(* CoDeSys 2.3 library: Util_plc.lib *)

(* Global variable list: Globale_Variablen *)
(*
 PLC1131-Library with various Utility-Functions:
 1. Bit_xx:		BOOL-Array-Pack, -Split and -Scan
 2. Hwio_xx:	DWORD/DINT-Array-Pack and -Split
 3. Tcs_xx:	Interface to System-Time/Timer and Run-Time-System-Specials
 4. Util_xx:		String/Character-Handling
 5. Mem_xx:	Marker/Memory-Area-Handling
 6. MSys_xx:	Interface to Settings and Information from MCore/MSys
 Copyright: G.Bachmann GmbH, 1996-1997, Feldkirch - Austria
*)
VAR_GLOBAL CONSTANT
	UTIL_PLC_LIBVER			  :	STRING(16) 	:=	'V1.40 Release';	(* Version String *)
	UTIL_PLC_MMPREADY         : BOOL        :=  TRUE;               (* MMP Ready *)

    (* Error-Return-Codes *)
    Tcs_ERC_ParmInvalid:		DINT := -2;			(* Parameters are invalid *)
    Tcs_ERC_NoSelf:				DINT := -8;			(* Caller is no PLC *)
    Tcs_ERC_Internal:           DINT := -11;		(* external function not supported *)

    (* constants for 'AreaCode' of Mem_GetSize and Mem_Clear *)
    Tcs_MX_Code:				DINT := 1;
    Tcs_MB_Code:				DINT := 2;
    Tcs_MD_Code:				DINT := 3;
    Tcs_MR_Code:				DINT := 4;
    Tcs_MW_Code:				DINT := 5;
    Tcs_RD_Code:				DINT := 19;
    Tcs_GD_Code:				DINT := 35;

    (* these constants occur in 'ConfState' of TCS_ARGINFO *)
    Tcs_CONF_PassString:		DINT := 16#40;		(* ArgumentStr="..." *)
    Tcs_CONF_PassNumber:		DINT := 16#80;		(* ArgumentNum=... *)
    Tcs_CONF_ReinitRetain:		DINT := 16#400;
    Tcs_CONF_MarkerBattPool:	DINT := 16#800;
    Tcs_CONF_OverTime:			DINT := 16#1000;	(* RunTime > IntervalTime *)
    Tcs_CONF_SevereOverTime:	DINT := 16#2000;	(* RunTime >> IntervalTime *)

    (* constants for 'VersType' in Tcs_ARG_GetConfig' *)
	Tcs_VER_Alpha:                DINT := 1;          (* Alpha-Version *)
	Tcs_VER_Beta:                 DINT := 2;          (* Beta-Version *)
	Tcs_VER_Release:              DINT := 3;          (* Release-Version *)

    (* constants for 'DirCode' of MSys_GetDirName *)
    MSys_DIR_System:			DINT := 1;
    MSys_DIR_Driver:			DINT := 2;
    MSys_DIR_Application:		DINT := 3;
    MSys_DIR_Temporary:			DINT := 4;
    MSys_DIR_NonVolatile:		DINT := 5;

   (* constants for 'ProcType' of MSys_GetCpuInfo *)
    MSys_CPU_80386:				DINT := 0;			(* ME203/CS200/ES200 .. *)
    MSys_CPU_80486:				DINT := 1;
    MSys_CPU_Pentium:			DINT := 2;			(* MP2xx .. *)
	MSys_CPU_Geode: 			DINT := 3; 			(* AMD Geode *)
	MSys_CPU_Pentium3:			DINT := 4;			(* MPC2xx *)
	MSys_CPU_Pentium4: 			DINT := 5;
	MSys_CPU_Atom: 				DINT := 7;

	(* constants for 'RebootReason' of MSys_GetCpuInfo *)
	WDOG_REB_UNKNOWN: 			DINT := 0;			(* unknown reboot *)
	WDOG_REB_POWERFAIL: 		DINT := 1;			(* Powerfail caused reboot *)
	WDOG_REB_PANIC:				DINT := 2;			(* Panic caused reboot *)
	WDOG_REB_WDOGKNOWN:			DINT := 3;			(* Watchdog caused known reboot *)
	WDOG_REB_WDOGUNKNOWN:		DINT := 4;			(* unknown Watchdog reboot *)

	(* Return values of profile functions *)
	PF_E_PARM		: DINT := 16#800A_0110; (* invalid parameter *)
	PF_E_NOFILE		: DINT := 16#800A_0111; (* file not found *)
	PF_E_FILEBIG	: DINT := 16#800A_0112; (* file too big *)
	PF_E_FILEEMPTY	: DINT := 16#800A_0113; (* file is empty *)
	PF_E_NOSEC		: DINT := 16#800A_0114; (* section not found *)
	PF_E_NOGRP		: DINT := 16#800A_0115; (* group not found *)
	PF_E_NOKEY		: DINT := 16#800A_0116; (* keyword not found *)
	PF_E_ENDFILE	: DINT := 16#800A_0117; (* end of file reached *)
	PF_E_NOSET		: DINT := 16#800A_0119; (* set not found *)
	PF_E_NOUNIT		: DINT := 16#800A_0120; (* uint not found *)

	PF_MODE_RELOAD_FILE : DINT := 1; (* Reload configuration file on next read/write *)
	PF_MODE_USE_FILE : DINT := 2; (* Use configuration file (reset of PF_MODE_USE_DEFAULTS) *)
	PF_MODE_USE_DEFAULTS : DINT := 3; (* Use default values ignore configuration file *)
	PF_MODE_FILE_LOADED : DINT := 4; (* Use values from cache, do not load configuration file *)

	(* Commands of Util_CallCFcn *)
	Util_CMD_GetFcnHandle:			DWORD := 0;  (* get function handle *)
	Util_CMD_CallCFcn:				DWORD := 1;  (* call C-function *)

	(* State of Util_CallCFcn *)
	Util_ERR_CallC_HandleInit:			DINT := 1;  (* FB is not initialized *)
	Util_ERR_CallC_HandleOk:			DINT := 0;  (* able to call funcition handle *)
	Util_ERR_CallC_FcnNotFound:			DINT := -1;  (* function not found *)
	Util_ERR_CallC_NoHandle:			DINT := -2;  (* no function handle *)
	Util_ERR_CallC_InvalidCmd:			DINT := -3;  (* invalid command *)
	Util_ERR_CallC_NoSelf:				DINT := -8;	 (* caller is no PLC *)
    Util_ERR_CallC_Internal:            DINT := -11; (* internal error *)

	Util_CallC_Mode_C:					DINT := 0;	 (* native C function *)
	Util_CallC_Mode_PLC:				DINT := 1;	 (* PLC C function from external library *)

	(* possible states of Util_GetSymValByName and Util_SetSymValByName *)
	Util_ERR_SymVal_Ok:					DINT := 0;  (* success/no error *)
	Util_ERR_SymVal_InvalidName: 		DINT := -1; (* invalid/to long symbol-name *)
	Util_ERR_SymVal_NoHandle: 			DINT := -2; (* symbol not found in symbol-table *)
	Util_ERR_SymVal_InvalidLength: 		DINT := -3; (* an invalid symbol-values length *)

	(* possible errors of MSys_WdogSet *)
	Util_ERR_WDogSet_Ok: 				DINT := 0;	(* watchdog successfully reconfigured *)
	Util_ERR_WDogSet_WDNotActive:		DINT := -1;	(* watchdog has not been activated *)
	Util_ERR_WDogSet_LowWTime:			DINT := -2;	(* specified watch-time is too low *)
	Util_ERR_WDogSet_HighWTime:			DINT := -3; (* specified watch-time is too high *)
	Util_ERR_WDogSet_ConfigErr:			DINT := -4;	(* error configureing watch-dog *)

	(* Modes of Util_LIST_Get *)
	Util_LIST_GetHead:					DINT := 1; (* get head of list *)
	Util_LIST_GetTail:					DINT := 2; (* get tail of list *)
	Util_LIST_GetById:					DINT := 3; (* get a element by ID *)

	(* Modes of Util_LIST_Insert *)
	Util_LIST_InsertHead:				DINT := 1; (* insert a element at head *)
	Util_LIST_InsertTail:				DINT := 2; (* insert a element at tail *)

	(* Modes of Util_LIST_Remove *)
	Util_LIST_RemoveAll:				DINT := 0; (* remove all list elements *)
	Util_LIST_RemoveHead:				DINT := 1; (* remove head element *)
	Util_LIST_RemoveTail:				DINT := 2; (* remove tail element *)

	(* Error Codes of List FBs *)
	Util_ERR_LstOk:					DINT := 0;	(* Call was OK *)
	Util_ERR_LstNoMem:				DINT := -1; (* unable to alloc needed memory *)
	Util_ERR_LstInvHandle:			DINT := -2; (* invalid list handle *)
	Util_ERR_LstListEmpty:			DINT := -3; (* list is empty *)
	Util_ERR_LstListFull:			DINT := -4; (* list is full *)
	Util_ERR_LstInvCmd:				DINT := -5; (* invalid command *)
	Util_ERR_LstNotFound:			DINT := -6; (* list element was not found *)

	(* Modes of Util date and time functions *)
	Util_DT_Mode_UTC:			    DINT := 0; (* UTC time *)
	Util_DT_Mode_Local:			    DINT := 1; (* Local time *)

	(* Sources of Util_GetClock *)
	Util_CLOCK_RealTime: 			DINT := 0; (* system wide realtime clock *)
	Util_CLOCK_Monotonic: 			DINT := 16#1; (* Monotonic system-wide clock *)
	Util_CLOCK_Ptp: 				DINT := 16#10; (* PTP timer *)
	Util_CLOCK_RtcNano:				DINT := 16#20; (* RTC sec. + nanosec. based on CpuClocks,
													  since 3.95 same as CLOCK_REALTIME *)

	(* Results of Util64 timestamp functions *)
	Util64_TIMESTAMP_Result_OK:				DINT := 0; (* UTC time *)
	Util64_TIMESTAMP_Result_Error:			DINT := -1; (* Error, usually a struct pointer is NULL *)
	Util64_TIMESTAMP_Result_Overflow:		DINT := -2; (* overflow of 64bit value *)
	Util64_TIMESTAMP_Result_Underflow:		DINT := -3; (* underflow of 64bit value *)
	Util64_TIMESTAMP_Result_Negative:		DINT := -4; (* negative value *)
	Util64_TIMESTAMP_Result_Invalid_Range:	DINT := -5; (* range of parameter is invalid *)
	Util64_TIMESTAMP_Result_Zero:			DINT := -6; (* resulting value is 0 *)

END_VAR

(* Data type *)
(* return-structure of MSys_GetCpuInfo *)
TYPE MSYS_CPUINFO
STRUCT
	RetCode			: DINT;							(*  Success (0) - or Error-Code (<0) *)
	CpuSwitch		: DWORD;						(* Position/Code of Cpu-Switches *)
	ProcNum			: UDINT;						(* Processor-Number *)
	CpuClock		: UDINT;						(* Rate of Cpu-Clock in MHz *)
	TickRate		: UDINT;						(* Tick-Rate (Ticks per Second) for Scheduling *)
	TimeSlice		: UDINT;						(* Time-Slice in Ticks for Scheduling *)
	TotalTicks		: UDINT;						(* Number of Ticks since Power-Up *)
	AuxClkRate		: UDINT;						(* Rate of auxiliary Clock *)
	RestartCount	: UDINT;						(* Number of Restarts since last Reset of NV-Ram *)
	DebugMode		: DWORD;						(* DebugMode from MCONFIG.INI *)
	SizeDRam		: UDINT;						(* Size of 'Main'-Memory *)
	SizeNVRam		: UDINT;						(* Size of Non-Volatile-Ram *)
	ProcType		: UDINT;						(* Processor Type 0=80386, 2=Pentium *)
	pExtCpuInfo		: POINTER TO MSYS_EXTCPUINFO; 	(* Pointer to extended CPU info *)
	pEthStatist		: POINTER TO MSYS_ETHSTAT; 		(* Pointer to Ethernet statistik *)
	EnableMMP       : BOOL;                         (* M1 Multi Processing (SMP) enabled *)
    HyperThreading  : BOOL;                         (* Hyper threading active *)
    NbOfCores       : BYTE;                         (* Number OF logical cores available FOR SMP *)
    ReservedCores   : BYTE;                         (* Number OF reserved cores *)
END_STRUCT
END_TYPE

(* Data type *)
TYPE MSYS_ETHSTAT :
STRUCT
	InOverloadCount		: UDINT;					(* Counter input data overloads *)
	OutOverloadCount	: UDINT;					(* Counter output data overloads *)
	BcOverloadCount		: UDINT;					(* Counter broadcast overloads *)
	InBytes100msPeak	: UDINT;					(* In bytes peak load in 100 ms *)
	BcBytes100msPeak	: UDINT;					(* Broadcast peak load in 100 ms *)
	OutBytes100msPeak	: UDINT;					(* Out bytes peak load in 100 ms *)
	StartTicks10ms		: ARRAY[1..10] OF UDINT;	(* Ticks at start counting *)
	InBytes10ms			: ARRAY[1..10] OF UDINT;	(* In bytes last 10 millisec *)
	BcBytes10ms			: ARRAY[1..10] OF UDINT;	(* Broadcast bytes last 10 ms *)
	OutBytes10ms		: ARRAY[1..10] OF UDINT;	(* Out bytes last 10 millisec *)
	CurrIndex100s		: UDINT;					(* Index to xx100s[] 0 .. 9 *)
	InPacks100s			: ARRAY[1..10] OF UDINT;	(* In packets last 100 seconds *)
	InBytes100s			: ARRAY[1..10] OF UDINT;	(* In bytes last 100 seconds *)
	BcPacks100s			: ARRAY[1..10] OF UDINT;	(* Broadcast packets last 100 s *)
	BcBytes100s			: ARRAY[1..10] OF UDINT;	(* Broadcast bytes last 100 s *)
	OutPacks100s		: ARRAY[1..10] OF UDINT;	(* Out packets last 100 seconds *)
	OutBytes100s		: ARRAY[1..10] OF UDINT;	(* Out bytes last 100 seconds *)
	InPacksTotal		: UDINT;					(* In packets since reboot *)
	InBytesTotalLow		: DWORD;					(* In bytes since reboot low DWORD *)
	InBytesTotalHigh	: DWORD;					(* In bytes since reboot high DWORD *)
	BcPacksTotal		: UDINT;					(* Broadcasts since reboot *)
	BcBytesTotalLow		: DWORD;					(* Broadcast bytes since reboot low DWORD *)
	BcBytesTotalHigh	: DWORD;					(* Broadcast bytes since reboot high DWORD *)
	OutPacksTotal		: UDINT;					(* Out packets since reboot *)
	OutBytesTotalLow	: DWORD;					(* Out bytes since reboot low DWORD *)
	OutBytesTotalHigh	: DWORD;					(* Out bytes since reboot high DWORD *)
END_STRUCT
END_TYPE

(* Data type *)
TYPE MSYS_EXTCPUINFO :
STRUCT
	CurrTemp: UDINT; (* Current CPU temperature in % *)
	MinTemp: UDINT; (* Minimum CPU temperature in % *)
	MaxTemp: UDINT; (* Maximum CPU temperature in % *)
	CpuUsage100Low: DWORD; (* Cpu Usage last 100 seconds low DWord *)
	CpuUsage100High: DWORD; (* Cpu Usage last 100 seconds high DWord *)
	CpuUsage1000Low: DWORD; (* Cpu Usage last 1000 seconds low DWord *)
	CpuUsage1000High: DWORD; (* Cpu Usage last 1000 seconds high DWord *)
	CpuUsageTotalLow: DWORD; (* Accumulated Cpu Time in Clocks low DWord *)
	CpuUsageTotalHigh: DWORD; (* Accumulated Cpu Time in Clocks high DWord *)
	TotalTimeLow: DWORD; (* Clocks since last reset (100%) low DWord *)
	TotalTimeHigh: DWORD; (* Clocks since last reset (100%) high DWord *)
	Spare: ARRAY [1..4] OF UDINT; (* NOT used, 0 FOR now *)
	UnitsTime: UDINT; (* Clocks per us (CPU MHz) *)
	LastIdleTime: UDINT; (* TIME in us Idle last ran *)
	MaxPccErases: UDINT; (* Maximum PC-Card erases *)
	MaxFlashErases: UDINT; (* Maximum Flash erases *)
	StrayInterrupts: UDINT; (* Number of stray interrupts *)
	SyncHigh: UDINT; (* Sync Rate fuer High in us *)
	SyncLow: UDINT; (* Sync Rate fuer Low in us *)
	pSyncCount: POINTER TO UDINT; (* Sync interrupts since boot *)
	pAuxClkCount: POINTER TO UDINT; (* Aux clocks since boot *)
	PccPresent: BYTE; (* PC-Card is present *)
	PccPluggedIn: BYTE; (* PC-Card is plugged in *)
	PccWritable: BYTE; (* No PC-Card write protection *)
	PccCheckError: BYTE; (* Error in boot check on PC-Card *)
	FlashPresent: BYTE; (* File Flash is present *)
	FlashWritable: BYTE; (* No Flash write protection *)
	FlashCheckError: BYTE; (* Error in boot check on Flash *)
	NVRamSupplError: BYTE; (* Error in NV-Ram supply *)
	NVRamCheckError: BYTE; (* Error in boot check on NV-Ram *)
	StackCheckError: BYTE; (* Stack overflow in one task *)
	DRamCheckError: BYTE; (* Checksum error in DRam *)
	RTCError: BYTE; (* Error in RTC value *)
    SoftBootError: BYTE; (* Soft boot error, M1 BY run *)
    HardBootError: BYTE; (* Hard boot error, booting aborted *)
    LongNameEnable: BYTE; (* Long filenames ON/OFF *)
    TickSource: BYTE; (* M_TICK_TIMER, M_TICK_RTC *)
    SntpTimestamp: DATE; (* SNTP TIME in sec. since 1970 *)
    (* Below here needs MSys 2.00 Release *)
	RebootReason: UDINT; (* reboot reason *)
	RebootInf: STRING(39); (* reboot info text *)
    (* Below here needs MSys 3.20 Release *)
    SntpTimeRecv: TIMESPEC; (* Last received SNTP TIME *)
    SntpTimeCorr: TIMESPEC; (* Last received SNTP TIME maybe
                               corrected by "SntpMaxCorrection"
                               and converted to local time. *)
    SntpMaxCorrection: DWORD; (* Maximum allowed change per
                                 SNTP update [sec]. *)
END_STRUCT
END_TYPE

(* Data type *)
(* return-structure of  Tcs_ARG_GetConfig *)
TYPE TCS_ARGINFO
STRUCT
    Verbose: DINT;                   (* Verbose/Debug-Level *)
    StopAfterStart: DINT;            (* indicates loading by gb-PLC/PS *)
    ConfState: DWORD;                (* (see 'Global Constants') *)
    TimeSlice: DINT;                 (* Interval-Time in 0.1 Milli-Seconds *)
    WithWatchdog: DINT;              (* 1 if Watchdog supervision, 0 otherwise *)
    WatchTime: DINT;                 (* Watchdog-Time *)
    MissingModules: DWORD;           (* BitMask of missing modules (first 31 only) *)
    ArgNumber: DINT;                 (* Number of setting 'ArgumentNum=' *)
    ArgStringLen: DINT;              (* Len of String of setting 'ArgumentStr=' *)
    Name: STRING(15);                (* Name of running Project / Module *)
    VersCode: ARRAY[1..3] OF UDINT;  (* version of current project/sw-module *)
	VersType: UDINT;                 (* version type (see 'global constants') *)
END_STRUCT
END_TYPE

(* Data type *)
(* return-structure of Tcs_RTC_LocalTime and Tcs_RTC_UTCTime *)
(* date+time in this format can be converted back to type DATE_AND_TIME
    by Tcs_RTC_BuildDT *)
TYPE TCS_CLOCK
STRUCT
    Second: DINT;		(* range 0 - 59 *)
    Minute: DINT;		(* range 0 - 59 *)
    Hour: DINT;			(* range 0 - 23 *)
    Day: DINT;			(* range 1 - 31 *)
    Month: DINT;		(* range 1 - 12 *)
    Year: DINT;			(* years since 1900 *)
    WeekDay: DINT;	    (* range 0 = Sunday ... 6 = Saturday *)
    YearDay: DINT;		(* range 0 - 365 *)
    DSTFlag: DINT;		(* DayLightSaving-Time Flag *)
END_STRUCT
END_TYPE

(* Data type *)
(* return-structure of Tcs_CYC_GetCycStat *)
TYPE TCS_CYCSTAT
STRUCT						(* all times in this structure are in ticks *)
    EntrySize: DINT;		(* size of this structure in bytes *)
    EntryType: DINT;		(* scaling of times to ticks (ticks per 0.1 Milli-Second) *)
    Running: DINT;			(* scaling of times to ticks (tick-duration in 0.1 Milli-Seconds *)
    Priority: DINT;			(* specified task priority *)
    CycTime: DWORD;			(* specified Interval-Time *)
    DiffTime: DWORD;		(* period between last two cycle-starts *)
    MinTime: DWORD;			(* min. DiffTime seen *)
    MaxTime: DWORD;			(* max. DiffTime seen *)
    AvgTime: DWORD;			(* average of DiffTime *)
    AvgParam: DWORD;		(* 32 *)
    CycCnt: DWORD;			(* counter of cycles *)
    Activity: DWORD;		(* reserved *)
    LastTime: DWORD;		(* time-stamp of last cycle *)
    MinRunTime: DWORD;		(* (only computed if CycTime > 0): min. of period of cycles *)
    MaxRunTime: DWORD;		(* (only computed if CycTime > 0): max. of period of cycles *)
    AvgRunTime: DWORD;		(* (only computed if CycTime > 0): avg. of period of cycles *)
	Running_us: DWORD;		(* tick-duration in micro-seconds, needs MSYS 2.02 or above *)
END_STRUCT
END_TYPE

(* Data type *)
TYPE TIMESPEC :
STRUCT
	DateAndTime: DT;
    NanoSeconds: UDINT;
END_STRUCT
END_TYPE

(* Data type *)
(* 64bit Timestamp split into DATE, TIME and NanoSeconds *)
TYPE UTIL64_DATETIME :
STRUCT
	DateValue  : DATE; (* DATE part of 64bit Timestamp *)
	TimeValue : TIME; (* TIME part of 64bit Timestamp *)
	NanoSeconds : UDINT; (* Nanosecons not contained in TimeValue *)
END_STRUCT
END_TYPE

(* Data type *)
(* 64bit Timestamp Value for time in nanoseconds *)
(* The value is unsigned *)
TYPE UTIL64_TIMESTAMP :
STRUCT
	TimestampNsLow  : DWORD; (* 4 byte little endian low part of 64bit *)
	TimestampNsHigh : DWORD; (* 4 byte little endian high part of 64bit *)
END_STRUCT
END_TYPE

(* Data type *)
(* return-structure of Util_GetCycStat *)
TYPE UTIL_CYCSTAT :
STRUCT
    Priority: DINT;			(* specified task priority [vxworks] *)
    CycTime: DWORD;			(* specified cycle-time [us] *)
	MainRatio: DWORD;		(* execution-rate of the task-POU *)
    CycCnt: DWORD;			(* counter of cycles *)
    RunTimeMin: DWORD;		(* Minimum Run Time in us *)
    RunTimeMax: DWORD;		(* Maximum Run Time in us *)
    RunTimeAvg: DWORD;		(* Average Run Time in us *)
	RunTimeTotal: DWORD;	(* Total run time in us *)
	CycleTimeMin: DWORD;    (* Minimum Cycle TIME in us *)
    CycleTimeMax: DWORD;    (* Maximum Cycle TIME in us *)
    CycleTimeAvg: DWORD;    (* Average Cycle TIME in us *)
	ErrorCode:  DINT;		(* OK/Done, Error-Code in case of error *)
END_STRUCT
END_TYPE

(* Data type *)
(* time structure TM *)
(* this time structure can be converted to DATE_AND_TIME (DT) *)
TYPE UTIL_TM
STRUCT
    Second: DINT;		(* range 0 - 59 *)
    Minute: DINT;		(* range 0 - 59 *)
    Hour: DINT;			(* range 0 - 23 *)
    Day: DINT;			(* range 1 - 31 *)
    Month: DINT;		(* range 1 - 12 *)
    Year: DINT;			(* years since 1900 *)
    WeekDay: DINT;	    (* range 0 = Sunday ... 6 = Saturday *)
    YearDay: DINT;		(* range 0 - 365 *)
    DSTFlag: DINT;		(* DayLightSaving-Time Flag *)
END_STRUCT
END_TYPE

(* POU BCD_TO_DINT, ST *)
(******************************************************************************
Description: Converts from BCD to Integer(32bit)
Input:
  - Num: BCD-value; Range 8 digits
Output:
    none
Return:
    Integer(32bit) value of BCD-value: Range 0 to 99999999
******************************************************************************)
FUNCTION BCD_TO_DINT : DINT
VAR_INPUT
	Num : DWORD;
END_VAR
;
END_FUNCTION

(* POU BCD_TO_INT, ST *)
(******************************************************************************
Description: Converts from BCD to Integer(16bit)
Input:
  - Num: BCD-value; Range 4 digits
Output:
    none
Return:
    Integer(16bit) value of BCD-value: Range 0 to 9999
******************************************************************************)
FUNCTION BCD_TO_INT : INT
VAR_INPUT
	Num : WORD;
END_VAR
;
END_FUNCTION

(* POU BCD_TO_SINT, ST *)
(******************************************************************************
Description: Converts from BCD to Integer(8bit)
Input:
  - Num: BCD-value; Range 2 digits
Output:
    none
Return:
    Integer(8bit) value of BCD-value: Range 0 to 99
******************************************************************************)
FUNCTION BCD_TO_SINT : SINT
VAR_INPUT
	Num : BYTE;
END_VAR
;
END_FUNCTION

(* POU Bit_FieldPack, IL *)
(******************************************************************************
Description: Packs Bits of the BOOL-Array to a DWORD-Array
Input:
  - StartAddrBits: Address of the BOOL array, use ADR() operator
  - StartIndx: Start index
  - EndIndx: End index
  - BitsTogether: Determines the number of Bits to pack together in a DWORD 
  - StartAddrPacked: Address of the DWORD-Array, use ADR() operator
Output:
  - StartAddrPacked: Moved bits from BOOL-Array
Return: Function checks if 'EndIndx'+1-'StartIndx' must is multiple 
    of 'BitsTogether'!
    - TRUE: Parameters are OK
    - FALSE: Wrong parameters
******************************************************************************)
FUNCTION Bit_FieldPack : BOOL
VAR_INPUT
	StartAddrBits: DWORD;
	StartIndx: DINT;
	EndIndx: DINT;
	BitsTogether: DINT;
	StartAddrPacked: DWORD;
END_VAR
	LD		0
END_FUNCTION

(* POU Bit_FieldScan, IL *)
(******************************************************************************
Description: Scans the BOOL-Array from StartIndx to EndIndx for the 
    first TRUE-Element
Input:
  - StartAddr: Address of BOOL array, use ADR() operator
  - StartIndx: Start index
  - EndIndx: End index
Output:
    none
Return: Index of the first TRUE element, or all zero
    - >= 0: Index of element
    - -1: no TRUE element is found
******************************************************************************)
FUNCTION Bit_FieldScan : DINT
VAR_INPUT
	StartAddr: DWORD;
	StartIndx: DINT;
	EndIndx: DINT;
END_VAR
LD 0
END_FUNCTION

(* POU Bit_FieldScanPack, IL *)
(******************************************************************************
Description: Packs Bits of the BOOL-Array to a DWORD-Array and scans for the
	last RUE element
Input:
  - StartAddrBits: Address of the BOOL array, use ADR() operator
  - StartIndx: Start index
  - EndIndx: End index
  - BitsTogether: Determines the number of Bits to pack together in a DWORD 
  - StartAddrPacked: Address of the DWORD-Array, use ADR() operator
Output:
  - StartAddrPacked: Moved bits from BOOL-Array
Return: Function checks if 'EndIndx'+1-'StartIndx' must is multiple 
    of 'BitsTogether'!
    - -2: Parameters are not OL
    - -1: No TRUE element is found
    - >= 0: Index of the last TRUE element
******************************************************************************)
FUNCTION Bit_FieldScanPack : DINT
VAR_INPUT
	StartAddrBits: DWORD;
	StartIndx: DINT;
	EndIndx: DINT;
	BitsTogether: DINT;
	StartAddrPacked: DWORD;
END_VAR
LD 0
END_FUNCTION

(* POU Bit_Pack, IL *)
(******************************************************************************
Description: Packs Bits of the BOOL-Array into a DWORD
Input:
  - StartAddr: Address of the BOOL array, use ADR() operator
  - NumberOf: Number of packing bits
Output:
    none
Return: Packed infomation of BOOL-array
*******************************************************************************)
FUNCTION Bit_Pack : DWORD
VAR_INPUT
	StartAddr: DWORD;
	NumberOf: DINT;
END_VAR
LD 0
END_FUNCTION

(* POU Bit_Split, IL *)
(******************************************************************************
Description: Unpacks Bits of a DWORD into a BOOL-Array
Input:
  - StartAddr: Address of the BOOL array, use ADR() operator
  - NumberOf: Number of depacking bits beginning at 0
  - Value: Packed Bits
Output:
  - StartAddr: This BOOL-array contains the unpacked bits of the DWORD
Return: Count equal to the set bits of the 'NumberOf'-Bits
*******************************************************************************)
FUNCTION Bit_Split : DINT
VAR_INPUT
	StartAddr: DWORD;
	NumberOf: DINT;
	Value: DWORD;
END_VAR
LD 0
END_FUNCTION

(* POU DINT_TO_BCD, ST *)
(******************************************************************************
Description: Converts from Integer(32bit) to BCD
Input:
  - Num: Integer(32bit) value; Range 0 to 99999999
Output:
    none
Return:
    BCD value; Range 8 digits
******************************************************************************)
FUNCTION DINT_TO_BCD : DWORD
VAR_INPUT
	Num : DINT;
END_VAR
;
END_FUNCTION

(* POU Hwio_Pack16, IL *)
(******************************************************************************
Description: Packs 16 values (type must be DWORD/DINT!) [set/clear] between 
    'StartAddr' and 'EndAddr' into a WORD (16bit)
Input:
  - StartAddr: Start address, use ADR() operator
  - EndAddr: End address, use ADR() operator
Output:
    none 
Return: WORD with packed bits
******************************************************************************)
FUNCTION Hwio_Pack16 : WORD
VAR_INPUT
    StartAddr: DWORD;
    EndAddr: DWORD; 
END_VAR
LD FALSE
END_FUNCTION

(* POU Hwio_Pack32, IL *)
(******************************************************************************
Description: Packs 32 values (type must be DWORD/DINT!) [set/clear] between 
    'StartAddr' and 'EndAddr' into a DWORD (32bit)
Input:
  - StartAddr: Start address, use ADR() operator
  - EndAddr: End address, use ADR() operator
Output:
    none 
Return: DWORD with packed bits
******************************************************************************)
FUNCTION Hwio_Pack32 : DWORD
VAR_INPUT
    StartAddr: DWORD;
    EndAddr: DWORD; 
END_VAR
LD FALSE
END_FUNCTION

(* POU Hwio_Pack8, IL *)
(******************************************************************************
Description: Packs 8 values (type must be DWORD/DINT!) [set/clear] between 
    'StartAddr' and 'EndAddr' into a DWORD (8bit)
Input:
  - StartAddr: Start address, use ADR() operator
  - EndAddr: End address, use ADR() operator
Output:
    none 
Return: BYTE with packed bits
******************************************************************************)
FUNCTION Hwio_Pack8 : BYTE
VAR_INPUT
    StartAddr: DWORD;
    EndAddr: DWORD; 
END_VAR
LD FALSE
END_FUNCTION

(* POU Hwio_Unpack, IL *)
(******************************************************************************
Description: Unpacking bits of a DWORD into a field of DWORDs [set/clear] 
Input:
  - StartAddr: Start address, use ADR() operator
  - EndAddr: End address, use ADR() operator
  - NumberOf: Number of unpacking bits
  - Packed: Value with packed bits
Output:
  - StartAddr to EndAddr: Unpacked bits
Return: If operation succeded
  - 0: Successful
  - Tcs_ERC_ParmInvalid: 'NumberOf' exceeds elements between 'Start'- 
    and 'EndAddr' 
******************************************************************************)
FUNCTION Hwio_Unpack : DINT
VAR_INPUT
    Packed: DWORD;  
    StartAddr: DWORD;
    EndAddr: DWORD; 
    NumberOf: DINT; 
END_VAR
LD FALSE
END_FUNCTION

(* POU INT_TO_BCD, ST *)
(******************************************************************************
Description: Converts from Integer(16bit) to BCD
Input:
  - Num: Integer(32bit) value; Range 0 to 9999
Output:
    none
Return:
    BCD value; Range 4 digits
******************************************************************************)
FUNCTION INT_TO_BCD : WORD
VAR_INPUT
	Num : INT;
END_VAR
;
END_FUNCTION

(* POU M100_PWMDutyCycleConv, ST *)
(******************************************************************************
Description: Converts a DutyCycle REAL to UINT.    
Input:
  - DutyCycle: with percent float value in range 0...100%
               Not fitting values will be limited to the valid range.
Output:
    none
Return:
	UINT converted DutyCycle. Value range. 0 .. 32768 (equals 100%)
******************************************************************************)
FUNCTION M100_PWMDutyCycleConv : WORD
VAR_INPUT
    DutyCycle : REAL;
END_VAR
;
END_FUNCTION

(* POU M100IO_GetCountedEvent, ST *)
(******************************************************************************
Description: splits a CountedEvent in its parts
Input:
  - Value: the current CountedEvent value to be split
Output:
  - State: state of the Event
  - Counter: how many times the event occured
  - NewEvent: true if the Counter changed since the last FB call
******************************************************************************)
FUNCTION_BLOCK M100IO_GetCountedEvent
VAR_INPUT
    Value : BYTE;
END_VAR
VAR_OUTPUT
	State : BOOL;
	Counter : WORD;
	NewEvent : BOOL;
END_VAR
VAR
	LastCounter : WORD;
END_VAR
;
END_FUNCTION_BLOCK

(* POU Mem_AtomicCopy, IL *)
(******************************************************************************
Description: Copy Memory-Area1 (Src) to Memory-Area2 (Dst) consistenly. All 
             reading and writing participants must use this function for a 
		     protection. 

Input:
  - Dst: Destination adress = Startadress of Memory-Area2
  - Src: Source adress = Start-adress of Memory-Area1 
  - Len: Length of the Memory-Area
Output:
    none 
Return: 
  - 0: Successful
  - Tcs_ERC_NoSelf: Caller is no PLC
  - Tcs_ERC_ParmInvalid: Parameters are invalid
******************************************************************************)
FUNCTION Mem_AtomicCopy : DINT
VAR_INPUT
	Dst: UDINT;
	Src: UDINT;
	Len: UDINT;
END_VAR
	LD		0
END_FUNCTION

(* POU Mem_Clear, IL *)
(******************************************************************************
Description: Clears the Memory/Marker-Area specified by 'AreaCode'
Input:
  - AreaCode: see CONSTANT variables Tcs_XX_Code, only this values are allowed
Output:
    none 
Return: Number of elements in the Area or error code
  - >= 0: Number of elements in the Area
  - -2: 'AreaCode' is invalid 
******************************************************************************)
FUNCTION Mem_Clear : DINT
VAR_INPUT
	AreaCode: DINT;
END_VAR
LD 0
END_FUNCTION

(* POU Mem_Copy, IL *)
(******************************************************************************
Description: Copy Memory-Area1 (Src) to Memory-Area2 (Dst)
Input:
  - Src: Source adress = Start-adress of Memory-Area1 
  - Dst: Destination adress = Startadress of Memory-Area2
  - Len: Length of the Memory-Area
Output:
    none 
Return: 
  -  0: Successful
  - -8: Caller is no PLC
******************************************************************************)
FUNCTION Mem_Copy : DINT
VAR_INPUT
	Dst: UDINT;
	Src: UDINT;
	Len: UDINT;
END_VAR
	LD		0
END_FUNCTION

(* POU Mem_GetSize, IL *)
(******************************************************************************
Description: Number of elements in the Memory/Marker-Area
Input:
  - AreaCode: see CONSTANT variables Tcs_xx_Code, only this values are allowed
Output:
    none 
Return: Number of elements in the Area or error code
  - >= 0: Number of elements in the Memory/Marker-Area
  - -2: 'AreaCode' is invalid 
******************************************************************************)
FUNCTION Mem_GetSize : DINT
VAR_INPUT
	AreaCode: DINT;
END_VAR
LD 0
END_FUNCTION

(* POU MSys_GetCpuInfo, IL *)
(******************************************************************************
Description: Fetching the system structure MSYS_CPUINFO
Input:
  - Dummy: meaningless
Output:
    none
Return:
    System structure MSYS_CPUINFO (see description in data types)
******************************************************************************)
FUNCTION MSys_GetCpuInfo : MSYS_CPUINFO
VAR_INPUT
	Dummy: DINT;
END_VAR
LD 0
END_FUNCTION

(* POU MSys_GetDirName, IL *)
(******************************************************************************
Description: Returns the path of the directory
Input:
  - DirCode: Code of directory
Output:
    none
Return:
    String of the system directory
******************************************************************************)
FUNCTION MSys_GetDirName : STRING(255)
VAR_INPUT
	DirCode: DINT;
END_VAR
LD 0
END_FUNCTION

(* POU MSys_GoPanic, ST *)
(******************************************************************************
Description: Initiate a System-Panic (SYS_APPPANIC)
Input:
  - Dummy: meaningless
Output:
    none
Return:
    meaningless
******************************************************************************)
FUNCTION MSys_GoPanic : DINT
VAR_INPUT
	Dummy: DINT;
END_VAR
;
END_FUNCTION

(* POU MSys_WdogSet, ST *)
(******************************************************************************
Description: reconfigures the watch-time of a projects software watch-dog,
             the watch-dog must have been activated

Note: be careful with applying a watch-time, 
	  the watch-time must have an adequate relation to the cycle-time and
      can cause reboots through the watch-dog if configured too low. 

Input:
  - WatchTime: watchdog-time, in milli- or micro-seconds
  - IsMicro: 0 - watch-time is in milli-seconds, 
             1 - watch-time is in micro-seconds
Return:
    zero on success or error-number otherwise
******************************************************************************)
FUNCTION MSys_WdogSet : DINT
VAR_INPUT
	WatchTime: UDINT;
	IsMicro: BOOL;
END_VAR
VAR
END_VAR
;
END_FUNCTION

(* POU MSys_WdogTrigger, ST *)
(******************************************************************************
Description: Trigger the software-watchdog of the PLC-project 
Input:
  - Dummy: meaningless
Output:
    none
Return:
    meaningless
******************************************************************************)
FUNCTION MSys_WdogTrigger : DINT
VAR_INPUT
	Dummy: DINT;
END_VAR
;
END_FUNCTION

(* POU Pf_Control, ST *)
(******************************************************************************
Description: Sets a specific mode of the Pf_Get and Pf_Set functions.    
Input:
  - Cmnd: mode to set (PF_MODE_XX)
Output:
    none
Return:
	>= 0 OK, line number (beginning at 0)
	< 0...error, see VAR_CONSTANT PF_E_XXX; convert this values with 
          DWORD_TO_DINT()
******************************************************************************)
FUNCTION Pf_Control : DINT
VAR_INPUT
	Cmnd	: DINT;
END_VAR
VAR
END_VAR
;
END_FUNCTION

(* POU pf_GetBool, ST *)
(******************************************************************************
Description: Reads a boolean value out of the specified file. Expression of 
    value in file has to be ON, OFF, YES, NO, TRUE, FALSE, 1 or 0. 
    Use this function in init section of PLC, it can take a little bit.    
Input:
  - Section: Name of section, 15 characters are significant, case sensitive. 
             If the string is empty it is used as a wildcard. 
  - Group: Name of group, 15 characters are significant, case sensitive. 
           If the string is empty it is used as a wildcard. 
  - Keyword: Name of keyword, 15 characters are significant, case sensitive
  - Default: Default Value, written to value when Keyword not found
  - Value: Returned value, use ADR() operator
  - StartLine: Start line of searching
  - FileName: file name, if an empty string is passed then in 'mconfig.ini' is searched
Output:
    none
Return:
	>= 0 OK, line number (beginning at 0)
	< 0...error, see VAR_CONSTANT PF_E_XXX; convert this values with 
          DWORD_TO_DINT()
******************************************************************************)
FUNCTION pf_GetBool : DINT
VAR_INPUT
	Section		: STRING;
	Group		: STRING;
	Keyword		: STRING;
	Default		: DINT;
	Value		: POINTER TO DINT;
	StartLine	: DINT;
	FileName	: STRING;
END_VAR
VAR
END_VAR
;
END_FUNCTION

(* POU pf_GetBoolExt, ST *)
(******************************************************************************
Description: Reads a boolean value out of the specified file. Expression of 
    value in file has to be ON, OFF, YES, NO, TRUE, FALSE, 1 or 0. 
    Use this function in init section of PLC, it can take a little bit.    
Input:
  - Section: 	Name of section, 15 characters are significant, case sensitive. 
             	If the string is empty it is used as a wildcard. 
  - Group: 		Name of group, 15 characters are significant, case sensitive. 
           	 	If the string is empty it is used as a wildcard. 
  - Set:     	Name of set, 15 characters are significant, case sensitive. 
             	If the string is empty it is used as a wildcard. 
  - Unit: 	 	Name of unit, 15 characters are significant, case sensitive. 
           	 	If the string is empty it is used as a wildcard. 
  - Keyword: 	Name of keyword, 15 characters are significant, case sensitive
  - Default: 	Default Value, written to value when Keyword not found
  - Value: 	 	Returned value, use ADR() operator
  - StartLine: 	Start line of searching
  - FileName: 	File name, if an empty string is passed then 'mconfig.ini' is used
Output:
    none
Return:
	>= 0 OK, line number (beginning at 0)
	< 0...error, see VAR_CONSTANT PF_E_XXX; convert this values with 
          DWORD_TO_DINT()
******************************************************************************)
FUNCTION pf_GetBoolExt : DINT
VAR_INPUT
	Section		: STRING;
	Group		: STRING;
	Set			: STRING;
	Unit		: STRING;
	Keyword		: STRING;
	Default		: DINT;
	Value		: POINTER TO DINT;
	StartLine	: DINT;
	FileName	: STRING;
END_VAR
VAR
END_VAR
;
END_FUNCTION

(* POU pf_GetInt, IL *)
(******************************************************************************
Description: Reads an integer value out of the specified file. 
    Use this function in init section of PLC, it can take a little bit.    
Input:
  - Section: Name of section, 15 characters are significant, case sensitive. 
             If the string is empty it is used as a wildcard. 
  - Group: Name of group, 15 characters are significant, case sensitive. 
           If the string is empty it is used as a wildcard. 
  - Keyword: Name of keyword, 15 characters are significant, case sensitive
  - Default: Default Value, written to value when Keyword not found
  - Value: Returned value, use ADR() operator
  - StartLine: Start line of searching
  - FileName: file name, if an empty string is passed then in 'mconfig.ini' is searched
Output:
    none
Return:
	>= 0 OK, line number (beginning at 0)
	< 0...error, see VAR_CONSTANT PF_E_XXX; convert this values with 
          DWORD_TO_DINT()
******************************************************************************)
FUNCTION pf_GetInt : DINT
VAR_INPUT
	Section		: STRING;
	Group		: STRING;
	Keyword		: STRING;
	Default		: DINT;
	Value		: POINTER TO DINT;
	StartLine	: DINT;
	FileName	: STRING;
END_VAR
VAR
END_VAR
	LD		0
END_FUNCTION

(* POU pf_GetIntExt, IL *)
(******************************************************************************
Description: Reads an integer value out of the specified file. 
    Use this function in init section of PLC, it can take a little bit.    
Input:
  - Section: 	Name of section, 15 characters are significant, case sensitive. 
             	If the string is empty it is used as a wildcard. 
  - Group: 		Name of group, 15 characters are significant, case sensitive. 
           	 	If the string is empty it is used as a wildcard. 
  - Set:     	Name of set, 15 characters are significant, case sensitive. 
             	If the string is empty it is used as a wildcard. 
  - Unit: 	 	Name of unit, 15 characters are significant, case sensitive. 
           	 	If the string is empty it is used as a wildcard. 
  - Keyword: 	Name of keyword, 15 characters are significant, case sensitive
  - Default: 	Default Value, written to value when Keyword not found
  - Value: 	 	Returned value, use ADR() operator
  - StartLine: 	Start line of searching
  - FileName: 	File name, if an empty string is passed then 'mconfig.ini' is used
Output:
    none
Return:
	>= 0 OK, line number (beginning at 0)
	< 0...error, see VAR_CONSTANT PF_E_XXX; convert this values with 
          DWORD_TO_DINT()
******************************************************************************)
FUNCTION pf_GetIntExt : DINT
VAR_INPUT
	Section		: STRING;
	Group		: STRING;
	Set			: STRING;
	Unit		: STRING;
	Keyword		: STRING;
	Default		: DINT;
	Value		: POINTER TO DINT;
	StartLine	: DINT;
	FileName	: STRING;
END_VAR
VAR
END_VAR
	LD		0
END_FUNCTION

(* POU pf_GetSecGrp, ST *)
(******************************************************************************
Description: returns the name of the preceding section and group of the passed-on
             line number. 

Input:
  - LastLine: the search starts from this line backwards. 
  - FileName: file name, if an empty string is passed then in 'mconfig.ini' is searched
Output:
  - Section: Name of section, 15 characters are significant, case sensitive
  - Group: Name of group, 15 characters are significant, case sensitive 
Return:
	>= 0 OK, line number (beginning at 0)
	< 0...error, see VAR_CONSTANT PF_E_XXX; convert this values with 
          DWORD_TO_DINT()
******************************************************************************)

FUNCTION pf_GetSecGrp : DINT
VAR_INPUT
	Section: STRING(15);
	Group: STRING(15);
	LastLine: DINT;
	FileName: STRING;
END_VAR
VAR
END_VAR
;
END_FUNCTION

(* POU Pf_GetStrg, ST *)
(******************************************************************************
Description: Reads a string value out of the specified file. 
    Use this function in init section of PLC, it can take a little bit.    
Input:
  - Section: Name of section, 15 characters are significant, case sensitive. 
             If the string is empty it is used as a wildcard. 
  - Group: Name of group, 15 characters are significant, case sensitive. 
           If the string is empty it is used as a wildcard. 
  - Keyword: Name of keyword, 15 characters are significant, case sensitive
  - Default: Default Value, written to value when Keyword not found  
  - Value: Returned value, max 80 characters
		   Important: String size has to be 80 chars !!
  - StartLine: Start line of searching
  - FileName: file name, if an empty string is passed then in 'mconfig.ini' is searched
Output:
    none
Return:
	>= 0 OK, line number (beginning at 0)
	< 0...error, see VAR_CONSTANT PF_E_XXX; convert this values with 
          DWORD_TO_DINT()
******************************************************************************)
FUNCTION Pf_GetStrg : DINT
VAR_INPUT
	Section		: STRING;
	Group		: STRING;
	Keyword		: STRING;
	Default		: STRING;
	Value		: STRING;
	StartLine	: DINT;
	FileName	: STRING;
END_VAR
VAR
END_VAR
;
END_FUNCTION

(* POU Pf_GetStrg2, ST *)
(******************************************************************************
Description: Reads a string value out of the specified file.
	This is the same function as Pf_GetStrg except for the max length of the 
    value sting.  
    Use this function in init section of PLC, it can take a little bit.    
Input:
  - Section: Name of section, 15 characters are significant, case sensitive. 
             If the string is empty it is used as a wildcard. 
  - Group: Name of group, 15 characters are significant, case sensitive. 
           If the string is empty it is used as a wildcard. 
  - Keyword: Name of keyword, 15 characters are significant, case sensitive
  - Default: Default Value, written to value when Keyword not found
  - Value: Returned value (not a default string)
		   Since M-Base 3.70 149 characters are supported. The maximum length of 
           Pf_GetStr2 is reduced by the length of the keyword and of the string " = ".
		   Important: String size has to be 255 chars !!
  - StartLine: Start line of searching
  - FileName: file name, if an empty string is passed then in 'mconfig.ini' is searched
Output:
    none
Return:
	>= 0 OK, line number (beginning at 0)
	< 0...error, see VAR_CONSTANT PF_E_XXX; convert this values with 
          DWORD_TO_DINT()
******************************************************************************)
FUNCTION Pf_GetStrg2 : DINT
VAR_INPUT
	Section		: STRING;
	Group		: STRING;
	Keyword		: STRING;
	Default		: STRING;
	Value		: STRING(255);
	StartLine	: DINT;
	FileName	: STRING;
END_VAR
VAR
END_VAR
;
END_FUNCTION

(* POU Pf_GetStrgExt, ST *)
(******************************************************************************
Description: Reads a string value out of the specified file. 
    Use this function in init section of PLC, it can take a little bit.    
Input:
  - Section: 	Name of section, 15 characters are significant, case sensitive. 
             	If the string is empty it is used as a wildcard. 
  - Group: 		Name of group, 15 characters are significant, case sensitive. 
           	 	If the string is empty it is used as a wildcard. 
  - Set:     	Name of set, 15 characters are significant, case sensitive. 
             	If the string is empty it is used as a wildcard. 
  - Unit: 	 	Name of unit, 15 characters are significant, case sensitive. 
           	 	If the string is empty it is used as a wildcard. 
  - Keyword: 	Name of keyword, 15 characters are significant, case sensitive
  - Default: 	Default Value, written to value when Keyword not found
  - Value: 	 	Returned value, use ADR() operator. 
                Important: String size has to be 255 chars !!
                Since M-Base 3.70 149 characters are supported. The maximum length of 
                Pf_GetStrgExt is reduced by the length of the keyword and of the string 
                " = ".
  - StartLine: 	Start line of searching
  - FileName: 	File name, if an empty string is passed then 'mconfig.ini' is used
Output:
    none
Return:
	>= 0 OK, line number (beginning at 0)
	< 0...error, see VAR_CONSTANT PF_E_XXX; convert this values with 
          DWORD_TO_DINT()
******************************************************************************)
FUNCTION Pf_GetStrgExt : DINT
VAR_INPUT
	Section		: STRING;
	Group		: STRING;
	Set			: STRING;
	Unit		: STRING;
	Keyword		: STRING;
	Default		: STRING;
	Value		: STRING(255);
	StartLine	: DINT;
	FileName	: STRING;
END_VAR
VAR
END_VAR
;
END_FUNCTION

(* POU Pf_SetStrg_NB, ST *)
(******************************************************************************
Description: Writes a string value in the specified file. The keywords value 
             can be edited only, it must exist already. This is a non-blocking 
             function. 
Input:
  - Req:  request-enable
  - Section: Name of section, 15 characters are significant, case sensitive. 
             If the string is empty it is used as a wildcard. 
  - Group: Name of group, 15 characters are significant, case sensitive. 
           If the string is empty it is used as a wildcard. 
  - Keyword: Name of keyword, 15 characters are significant, case sensitive
  - Value: value, max 255 characters (the Core components of MBASE 3.50 support 
           max. 80 characters for the whole line of the keyword entry).
		   Since M-Base 3.70 149 characters are supported. The maximum length of 
           Pf_SetStrg_NB is reduced by the length of the keyword and of the string " = ".
  - StartLine: Start line of searching
  - FileName: file name, if an empty string is passed then in 'mconfig.ini' is searched
Output:
  - Done:  TRUE => operation completed 
  - Error:  TRUE in case of error 
  - Status:  0: OK/Done, 1: BUSY, Error-Code in case of error 
    (see VAR_CONSTANT PF_E_XXX; convert this values with DWORD_TO_DINT())
  - WrittenLine: written line number (beginning at 0)

******************************************************************************)
FUNCTION_BLOCK Pf_SetStrg_NB
VAR_INPUT
	Req         : BOOL;
	Section     : STRING;
	Group       : STRING;
	Keyword		: STRING;
	Value       : STRING(255);
	StartLine   : DINT;
	FileName    : STRING;
END_VAR
VAR_OUTPUT
	Done        : BOOL;
	Error       : BOOL;
	Status      : DINT;
    WrittenLine : UDINT;
END_VAR
VAR
    Pltd        : DWORD;
END_VAR
;
END_FUNCTION_BLOCK

(* POU Pf_SetStrgExt_NB, ST *)
(******************************************************************************
Description: Writes a string value in the specified file. The keywords value 
             can be edited only, it must exist already. This is a non-blocking 
             function. 
Input:
  - Req:  		request-enable
  - Section: 	Name of section, 15 characters are significant, case sensitive. 
             	If the string is empty it is used as a wildcard. 
  - Group: 		Name of group, 15 characters are significant, case sensitive. 
           	 	If the string is empty it is used as a wildcard. 
  - Set:     	Name of set, 15 characters are significant, case sensitive. 
             	If the string is empty it is used as a wildcard. 
  - Unit: 	 	Name of unit, 15 characters are significant, case sensitive. 
           	 	If the string is empty it is used as a wildcard. 
  - Keyword: 	Name of keyword, 15 characters are significant, case sensitive
  - Value: 		value, max 255 characters (the Core components of MBASE 3.50 support 
           		max. 80 characters for the whole line of the keyword entry)
 		        Since M-Base 3.70 149 characters are supported. The maximum length of 
                Pf_SetStrgExt_NB is reduced by the length of the keyword and of the 
                string " = ".
  - StartLine: 	Start line of search
  - FileName: 	file name, if an empty string is passed then 'mconfig.ini' is used
Output:
  - Done:  		TRUE => operation completed 
  - Error:  	TRUE in case of error 
  - Status:  	0: OK/Done, 1: BUSY, Error-Code in case of error 
			    (see VAR_CONSTANT PF_E_XXX; convert this values with DWORD_TO_DINT())
  - WrittenLine: written line number (beginning at 0)

******************************************************************************)
FUNCTION_BLOCK Pf_SetStrgExt_NB
VAR_INPUT
	Req         : BOOL;
	Section     : STRING;
	Group       : STRING;
	Set			: STRING;
	Unit		: STRING;
	Keyword		: STRING;
	Value       : STRING(255);
	StartLine   : DINT;
	FileName    : STRING;
END_VAR
VAR_OUTPUT
	Done        : BOOL;
	Error       : BOOL;
	Status      : DINT;
    WrittenLine : UDINT;
END_VAR
VAR
    Pltd        : DWORD;
END_VAR
;
END_FUNCTION_BLOCK

(* POU RTC_GetClock, ST *)
(******************************************************************************
Description: Gets the current time value of the system clock.
             This routine returns the system clock in seconds since 1970-01-01.
             The returned value is either UTC or LOCAL time, depending on 
             configured system time base.

Input:
  - Dummy: meaningless
Output:
    none
Return:
  - TIMESPEC structure (seconds + nanosecond part)
******************************************************************************)

FUNCTION RTC_GetClock : TIMESPEC
VAR_INPUT
	dummy: BOOL;
END_VAR
VAR
END_VAR
;
END_FUNCTION

(* POU SINT_TO_BCD, ST *)
(******************************************************************************
Description: Converts from Integer(8bit) to BCD
Input:
  - Num: Integer(32bit) value; Range 0 to 99
Output:
    none
Return:
    BCD value; Range 2 digits
******************************************************************************)
FUNCTION SINT_TO_BCD : BYTE
VAR_INPUT
	Num : SINT;
END_VAR
;
END_FUNCTION

(* POU Tcs_ARG_GetArgString, IL *)
(******************************************************************************
Description: Returns the String set with 'ArgumentStr=' (see file MCONFIG.INI)
Input:
  - Dummy: meaningless
Output:
    none
Return:
    String of Parameter 'ArgumentStr=' in file MCONFIG.INI
******************************************************************************)
FUNCTION Tcs_ARG_GetArgString : STRING(255)
VAR_INPUT
    Dummy: DINT;
END_VAR
LD FALSE
END_FUNCTION

(* POU Tcs_ARG_GetConfig, IL *)
(******************************************************************************
Description: Returns the system structure TCS_ARGINFO 
Input:
  - Dummy: meaningless
Output:
    none
Return:
    System Structure TCS_ARGINFO of current CPU (not all fields meaningful)
*****************************************************************************)
FUNCTION Tcs_ARG_GetConfig : TCS_ARGINFO
VAR_INPUT
    Dummy: DINT;
END_VAR
LD FALSE
END_FUNCTION

(* POU Tcs_CYC_GetCycStat, IL *)
(******************************************************************************
Description: Gets a copy of CYCSTAT-data. Deprecated support for the 
             first-task only since multitasking-environment (MSYS 3.80 R). 
             Multitasking is supported by Util_GetCycStat(). 
Input:
  - Dummy: meaningless
Output:
    none
Return:
  - TCS_CYCSTAT structure
******************************************************************************)
FUNCTION Tcs_CYC_GetCycStat: TCS_CYCSTAT
VAR_INPUT
    Dummy: DINT;
END_VAR
	LD		FALSE
END_FUNCTION

(* POU Tcs_CYC_GetMainRatio, IL *)
(******************************************************************************
Description: Returns Ratio of Intervals of Cyclic-Task(PLC_TASK) and SPS-Cycle. 
             Deprecated support for the first-task only since multitasking- 
             environment (MSYS 3.80 R). Multitasking is supported by 
             Util_GetCycStat(). 
Input:
  - Dummy: meaningless
Output:
    none
Return:
  - Tcs_CYC_GetMainRatio structure
******************************************************************************)
FUNCTION Tcs_CYC_GetMainRatio: DINT
VAR_INPUT
    Dummy: DINT;
END_VAR
	LD		FALSE
END_FUNCTION

(* POU Tcs_CYC_ReinitCycStat, IL *)
(******************************************************************************
Description: Reinit CYCSTAT-data
Input:
  - Dummy: meaningless
Output:
    none
Return:
    meaningless
******************************************************************************)
FUNCTION Tcs_CYC_ReinitCycStat: DINT
VAR_INPUT
    Dummy: DINT;
END_VAR
	LD		FALSE
END_FUNCTION

(* POU Tcs_CYC_SetCycStat, IL *)
(******************************************************************************
Description: Sets CYCSTAT/INTERVAL-data. Deprecated support for the 
             first-task only since multitasking-environment (MSYS 3.80 R).
             Multitasking is supported by Util_SetCycStat(). 
Input:
  - CycTime: PLC Interval Time in Ticks 
  - MainRatio: Ratio of PLC Interval Time to Task Interval Time
  - Priority: VxWorks Priority between 16 and 255
Output:
    none
Return: 
    meaningless
******************************************************************************)
FUNCTION Tcs_CYC_SetCycStat: DINT
VAR_INPUT
    CycTime: DWORD;
    MainRatio: DINT;
    Priority: DINT;
END_VAR
	LD		FALSE
END_FUNCTION

(* POU Tcs_EXC_Check, IL *)
(******************************************************************************
Description: Test Exception-Restart
Input:
  - Dummy: meaningless
Output:
    none
Return: Result of Exception-Restart
  - 1: Exception-Restart has been performed
  - else: not performed
*****************************************************************************)
FUNCTION Tcs_EXC_Check: DINT
VAR_INPUT
    Dummy: DINT;
END_VAR
LD FALSE
END_FUNCTION

(* POU Tcs_OLC_Check, IL *)
(******************************************************************************
Description: Test if an online change has been performed
Input:
  - Dummy: meaningless
Output:
    none
Return: Result of testing online change
  - 1: Online change has been performed
  - else: not performed
*****************************************************************************)
FUNCTION Tcs_OLC_Check: DINT
VAR_INPUT
    Dummy: DINT;
END_VAR
LD FALSE
END_FUNCTION

(* POU Tcs_RTC_BuildDT, IL *)
(******************************************************************************
Description: Converts TCS_CLOCK to DT-value according to local time zone
Input:
  - Clock: Time in format of TCS_CLOCK
Output:
    none
Return: 
    Time of format DATE_AND_TIME 
******************************************************************************)
FUNCTION Tcs_RTC_BuildDT: DATE_AND_TIME
VAR_INPUT
    Clock: TCS_CLOCK;
END_VAR
LD FALSE
END_FUNCTION

(* POU Tcs_RTC_GetDateAndTime, IL *)
(******************************************************************************
Description: Gets the current system date & time.
             This routine returns the current system time in either UTC or 
             LOCAL time, depending on configured system time base.

             ATTENTION: This function is deprecated. Please use 
                        function Util_RTC_GetDateAndTime instead 
                        of this function.

Input:
  - Dummy: meaningless
Output:
    none
Return: 
    Current date and time in DATE_AND_TIME format
******************************************************************************)
FUNCTION Tcs_RTC_GetDateAndTime: DATE_AND_TIME
VAR_INPUT
    Dummy: DINT;
END_VAR
LD FALSE
END_FUNCTION

(* POU Tcs_RTC_GetTime, IL *)
(******************************************************************************
Description: Get a monotonous time in microsecond resolution.
             This routine returns 'm_GetProcTime()' internally.
Input:
  - Dummy: meaningless
Output:
    none
Return: 
    Monotonous time
******************************************************************************)
FUNCTION Tcs_RTC_GetTime : UDINT
VAR_INPUT
    Dummy: DINT;
END_VAR
LD FALSE
END_FUNCTION

(* POU Tcs_RTC_LocalTime, IL *)
(******************************************************************************
Description: Converts DT to TCS_CLOCK according to local time zone
             (the local time-zone is considered since MSYS 3.10 R and 
             a compatibility-mode of >= 3.10)

             ATTENTION: This function is deprecated. Please use 
                        function Util_RTC_GetDateAndTime instead 
                        of this function.

Input:
  - D: Time of format DATE_AND_TIME
Output:
    none
Return: 
    Structure TCS_CLOCK
******************************************************************************)
FUNCTION Tcs_RTC_LocalTime: TCS_CLOCK
VAR_INPUT
    D: DATE_AND_TIME;
END_VAR
	LD		FALSE
END_FUNCTION

(* POU Tcs_RTC_SetDateAndTime, IL *)
(******************************************************************************
Description: Sets the current system date & time.
             This routine sets the system time to the value specified. Given
             time represents UTC or LOCAL time, depending on configured system
             timebase.

             ATTENTION: This function is deprecated. Please use 
                        function Util_RTC_SetDateAndTime instead 
                        of this function.

Input:
  - D: Date and Time of format DATE_AND_TIME 
Output:
    none
Return: Info of the action
  - 0: OK
  - 1: BUSY
  - else: ErrorCode
******************************************************************************)
FUNCTION Tcs_RTC_SetDateAndTime: DINT
VAR_INPUT
    D: DATE_AND_TIME;
END_VAR
LD FALSE
END_FUNCTION

(* POU Tcs_RTC_UTCTime, IL *)
(******************************************************************************
Description: Converts DT to TCS_CLOCK according to universal time zone (UTC)

             ATTENTION: This function is deprecated. Please use 
                        function Util_RTC_GetDateAndTime instead 
                        of this function.

Input:
  - D: Date and Time of format DATE_AND_TIME 
Output:
    none
Return: 
    Date and Time of format TCS_CLOCK
******************************************************************************)
FUNCTION Tcs_RTC_UTCTime: TCS_CLOCK
VAR_INPUT
    D: DATE_AND_TIME; 
END_VAR
LD FALSE
END_FUNCTION

(* POU Util64_ARRAY_TO_TIMESTAMP, ST *)
(******************************************************************************
Description: Converts from BYTE ARRAY[1..8] to 64bit Timestamp.    
Input:
  - TimestampNs: 8 Byte Array with little endian Timestamp raw data
  - TimestampResult: pointer to UTIL64_TIMESTAMP structure to be filled with
                     the result
Output:
    none
Return: DINT
	 0: Success (Util64_TIMESTAMP_Result_OK)
	-1: Error (Util64_TIMESTAMP_Result_Error)
	-6: timestamp is 0 (Util64_TIMESTAMP_Result_Zero)
******************************************************************************)
FUNCTION Util64_ARRAY_TO_TIMESTAMP : DINT
VAR_INPUT
	TimestampNs : ARRAY[1..8] OF BYTE;
	TimestampResult : POINTER TO UTIL64_TIMESTAMP;
END_VAR
;
END_FUNCTION

(* POU Util64_DATETIME_TO_TIMESTAMP, ST *)
(******************************************************************************
Description: Converts from DATE, TIME and ns to 64bit Timestamp.    
Input:
  - DateTime: a structure containing DATE, TIME and nanosecond part
  - TimestampResult: pointer to UTIL64_TIMESTAMP structure to be filled with
                     the result
Output:
    none
Return: DINT
	 0: Success (Util64_TIMESTAMP_Result_OK)
	-1: Error (Util64_TIMESTAMP_Result_Error)
	-2: NanoSeconds have invalid range (Util64_TIMESTAMP_Result_Invalid_Range)
******************************************************************************)
FUNCTION Util64_DATETIME_TO_TIMESTAMP : DINT
VAR_INPUT
	DateTime : UTIL64_DATETIME;
	TimestampResult : POINTER TO UTIL64_TIMESTAMP;
END_VAR
;
END_FUNCTION

(* POU Util64_ECTIME_TO_TIMESTAMP, ST *)
(******************************************************************************
Description: Converts from Ethercat DC-Time to 64bit Timestamp.    
Input:
  - ECTime: 64bit Timestamp structure containing nanoseconds since year 2000
  - TimestampResult: pointer to UTIL64_TIMESTAMP structure to be filled with
                     the result
Output:
    none
Return: DINT
	 0: Success (Util64_TIMESTAMP_Result_OK)
	-1: Error (Util64_TIMESTAMP_Result_Error)
	-2: Overflow (Util64_TIMESTAMP_Result_Overflow)
******************************************************************************)
FUNCTION Util64_ECTIME_TO_TIMESTAMP : DINT
VAR_INPUT
	ECTime : UTIL64_TIMESTAMP;
	TimestampResult : POINTER TO UTIL64_TIMESTAMP;
END_VAR
;
END_FUNCTION

(* POU Util64_LREAL_TO_TIMESTAMP, ST *)
(******************************************************************************
Description: Converts from LREAL to unsigned 64bit Timestamp.    
Input:
  - TimeNs: double float with nanoseconds in form of LREAL
  - TimestampResult: pointer to UTIL64_TIMESTAMP structure to be filled with
                     the result
Output:
    none
Return: DINT
	0 : Success (Util64_TIMESTAMP_Result_OK)
	-1: Error (Util64_TIMESTAMP_Result_Error)
	-2: Overflow (Util64_TIMESTAMP_Result_Overflow)
	-4: TimeNs is neagtive (Util64_TIMESTAMP_Result_Negative)
******************************************************************************)
FUNCTION Util64_LREAL_TO_TIMESTAMP : DINT
VAR_INPUT
	TimeNs : LREAL;
	TimestampResult : POINTER TO UTIL64_TIMESTAMP;
END_VAR
;
END_FUNCTION

(* POU Util64_TIMESPEC_TO_TIMESTAMP, ST *)
(******************************************************************************
Description: Converts from TIMESPEC to 64bit Timestamp.    
Input:
  - Timespec: TIMESPEC structure containing DT and nanoseconds
  - TimestampResult: pointer to UTIL64_TIMESTAMP structure to be filled with
                     the result
Output:
    none
Return: DINT
	 0: Success (Util64_TIMESTAMP_Result_OK)
	-1: Error (Util64_TIMESTAMP_Result_Error)
******************************************************************************)
FUNCTION Util64_TIMESPEC_TO_TIMESTAMP : DINT
VAR_INPUT
	Timespec : TIMESPEC;
	TimestampResult : POINTER TO UTIL64_TIMESTAMP;
END_VAR
;
END_FUNCTION

(* POU Util64_TIMESTAMP_ADD, ST *)
(******************************************************************************
Description: adds two unsigned 64bit Timestamps. 
Input:
  - TimeNs1: timestamp structure containing nanoseconds
  - TimeNs2: timestamp structure containing nanoseconds
  - TimestampResult: pointer to UTIL64_TIMESTAMP structure to be filled with
                     the result
Output:
    none
Return: DINT
	 0: Success (Util64_TIMESTAMP_Result_OK)
	-1: Error (Util64_TIMESTAMP_Result_Error)
	-2: Overflow (Util64_TIMESTAMP_Result_Overflow)
******************************************************************************)
FUNCTION Util64_TIMESTAMP_ADD : DINT
VAR_INPUT
	TimeNs1 : UTIL64_TIMESTAMP;
	TimeNs2 : UTIL64_TIMESTAMP;
	TimestampResult : POINTER TO UTIL64_TIMESTAMP;
END_VAR
;
END_FUNCTION

(* POU Util64_TIMESTAMP_ADD_Ext, ST *)
(******************************************************************************
Description: adds durations to a 64bit Timestamp structure.
             The Duration values can also be negative.
Input:
  - TimeNs1: timestamp structure containing nanoseconds
  - DurationHours: absolute amount of hours to add
                   accepted range -876000 to 876000 (approx. 100 years)
  - DurationMinutes: absolute amount of minutes to add
                     accepted range -5256000 to 5256000 (approx. 10 years)
  - DurationSeconds: absolute amount of seconds to add
                     accepted range -31536000 to 31536000 (approx. 1 year)
  - DurationMiliseconds: absolute amount of miliseconds to add
  - DurationNanoseconds: absolute amount of nanoseconds to add

  - TimestampResult: pointer to UTIL64_TIMESTAMP structure to be filled with
                     the result
Output:
    none
Return: DINT
	 0: Success (Util64_TIMESTAMP_Result_OK)
	-1: Error (Util64_TIMESTAMP_Result_Error)
	-2: Overflow (Util64_TIMESTAMP_Result_Overflow)
	-3: Underflow (Util64_TIMESTAMP_Result_Underflow)
	-5: Invalid Range of Durations (Util64_TIMESTAMP_Result_Invalid_Range)
******************************************************************************)
FUNCTION Util64_TIMESTAMP_ADD_Ext : DINT
VAR_INPUT
	TimeNs1 : UTIL64_TIMESTAMP;
	DurationHours : DINT;
	DurationMinutes : DINT;
	DurationSeconds : DINT;
	DurationMiliseconds : DINT;
	DurationNanoseconds : DINT;
	TimestampResult : POINTER TO UTIL64_TIMESTAMP;
END_VAR
;
END_FUNCTION

(* POU Util64_TIMESTAMP_EQ, ST *)
(******************************************************************************
Description: Compare two 64bit timestamps for equality
Input:
  - Timestamp1: 1nd timestamp for comparison (UTIL64_TIMESTAMP)
  - Timestamp2: 2nd timestamp for comparison (UTIL64_TIMESTAMP)
Output:
   none
Return: BOOL
   TRUE:  Timestamp1 == Timestamp2
   FALSE: Otherwise
******************************************************************************)
FUNCTION Util64_TIMESTAMP_EQ : BOOL
VAR_INPUT
	Timestamp1 : UTIL64_TIMESTAMP;
	Timestamp2 : UTIL64_TIMESTAMP;
END_VAR
VAR
END_VAR
;
END_FUNCTION

(* POU Util64_TIMESTAMP_GE, ST *)
(******************************************************************************
Description: Compare two 64bit timestamps to greater than or equal to
Input:
  - Timestamp1: 1st timestamp for comparison (UTIL64_TIMESTAMP)
  - Timestamp2: 2nd timestamp for comparison (UTIL64_TIMESTAMP)
Output:
   none
Return: BOOL
   TRUE:  Timestamp1 >= Timestamp2
   FALSE: Otherwise
******************************************************************************)
FUNCTION Util64_TIMESTAMP_GE : BOOL
VAR_INPUT
	Timestamp1 : UTIL64_TIMESTAMP;
	Timestamp2 : UTIL64_TIMESTAMP;
END_VAR
VAR
END_VAR
;
END_FUNCTION

(* POU Util64_TIMESTAMP_GT, ST *)
(******************************************************************************
Description: Compare two 64bit timestamps to greater than
Input:
  - Timestamp1: 1st timestamp for comparison (UTIL64_TIMESTAMP)
  - Timestamp2: 2nd timestamp for comparison (UTIL64_TIMESTAMP)
Output:
   none
Return: BOOL
   TRUE:  Timestamp1 > Timestamp2
   FALSE: Otherwise
******************************************************************************)
FUNCTION Util64_TIMESTAMP_GT : BOOL
VAR_INPUT
	Timestamp1 : UTIL64_TIMESTAMP;
	Timestamp2 : UTIL64_TIMESTAMP;
END_VAR
VAR
END_VAR
;
END_FUNCTION

(* POU Util64_TIMESTAMP_LE, ST *)
(******************************************************************************
Description: Compare two 64-bit timestamps to less than or equal to
Input:
  - Timestamp1: 1st timestamp for comparison (UTIL64_TIMESTAMP)
  - Timestamp2: 2nd timestamp for comparison (UTIL64_TIMESTAMP)
Output:
   none
Return: BOOL
   TRUE:  Timestamp1 <= Timestamp2
   FALSE: Otherwise
******************************************************************************)
FUNCTION Util64_TIMESTAMP_LE : BOOL
VAR_INPUT
	Timestamp1 : UTIL64_TIMESTAMP;
	Timestamp2 : UTIL64_TIMESTAMP;
END_VAR
VAR
END_VAR
;
END_FUNCTION

(* POU Util64_TIMESTAMP_LT, ST *)
(******************************************************************************
Description: Compare two 64bit timestamps on less than
Input:
  - Timestamp1: 1st timestamp for comparison (UTIL64_TIMESTAMP)
  - Timestamp2: 2nd timestamp for comparison (UTIL64_TIMESTAMP)
Output:
   none
Return: BOOL
   TRUE:  Timestamp1 < Timestamp2
   FALSE: Otherwise
******************************************************************************)
FUNCTION Util64_TIMESTAMP_LT : BOOL
VAR_INPUT
	Timestamp1 : UTIL64_TIMESTAMP;
	Timestamp2 : UTIL64_TIMESTAMP;
END_VAR
VAR
END_VAR
;
END_FUNCTION

(* POU Util64_TIMESTAMP_SUB, ST *)
(******************************************************************************
Description: substracts two unsigned 64bit Timestamps into a 64bit Timestamp. 

Input:
  - TimeNsMinuend: timestamp structure to subtract from
  - TimeNsSubtrahend: timestamp structure that is substracted

  - TimestampResult: pointer to UTIL64_TIMESTAMP structure to be filled with
                     the result
 Output:
    none
Return: DINT
	 0: Success (Util64_TIMESTAMP_Result_OK)
	-1: Error (Util64_TIMESTAMP_Result_Error)
	-3: Negative, the return value has to be negated 
       (Util64_TIMESTAMP_Result_Negative)
******************************************************************************)
FUNCTION Util64_TIMESTAMP_SUB : DINT
VAR_INPUT
	TimeNsMinuend : UTIL64_TIMESTAMP;
	TimeNsSubtrahend : UTIL64_TIMESTAMP;
	TimestampResult : POINTER TO UTIL64_TIMESTAMP;
END_VAR
;
END_FUNCTION

(* POU Util64_TIMESTAMP_SUB_Ext, ST *)
(******************************************************************************
Description: substracts two 64bit Timestamp structures to get durations.
             The durations can be negative.
Input:
  - TimeNsMinuend: unsigned timestamp structure to subtract from
  - TimeNsSubtrahend: unsigned timestamp structure that is substracted
  - calcAbsoluteDurations: if TRUE each duration value contains the full
    difference, except for DurationNanoseconds which then is relative to the 
    DurationSeconds value (to avoid overflow).
    Each Duration has the full DINT value range. Overflow is possible.
    If FALSE (default) each value is realtive, meaning all durations need to be
	added up for the full duration. The maximum for minutes or seconds is 59,
    respectively -59, for miliseconds +/-999 and nanoseconds +/-999999.
Output:
  - DurationHours: resulting amount of hours 
  - DurationMinutes: resulting amount minutes (relative to hours or absolute)
  - DurationSeconds: resulting amount seconds (relative to minutes or absolute)
  - DurationMiliseconds: resulting amount miliseconds
	(relative to seconds or absolute in which case be careful with overflow)
  - DurationNanoseconds: resulting amount nanoseconds
    (relative to miliseconds or in absolute case realtive so seconds)
******************************************************************************)
FUNCTION_BLOCK Util64_TIMESTAMP_SUB_Ext
VAR_INPUT
	TimeNsMinuend : UTIL64_TIMESTAMP;
	TimeNsSubtrahend : UTIL64_TIMESTAMP;
	calcAbsoluteDurations : BOOL;
END_VAR
VAR_OUTPUT
	DurationHours : DINT;
	DurationMinutes : DINT;
	DurationSeconds : DINT;
	DurationMiliseconds : DINT;
	DurationNanoseconds : DINT;
END_VAR
VAR_IN_OUT
END_VAR
VAR
END_VAR
;
END_FUNCTION_BLOCK

(* POU Util64_TIMESTAMP_TO_ARRAY, ST *)
(******************************************************************************
Description: Converts from 64bit Timestamp to an 8 Byte Array.    
Input:
  - TimestampNs: 64bit Timestamp structure
Output:
    none
Return:
	8 Byte Array with little endian Timestamp raw data.
******************************************************************************)
FUNCTION Util64_TIMESTAMP_TO_ARRAY : ARRAY[1..8] OF BYTE
VAR_INPUT
	TimestampNs : UTIL64_TIMESTAMP;
END_VAR
;
END_FUNCTION

(* POU Util64_TIMESTAMP_TO_DATETIME, ST *)
(******************************************************************************
Description: Converts from 64bit Timestamp to DATE, TIME and ns.    
Input:
  - Timestamp: 64bit Timestamp structure containing nanoseconds since year 1970
  - DateTimeResult: pointer to result structure containing DATE, TIME and
                    nanosecond part
Output:
    none
Return: DINT
	 0: Success (Util64_TIMESTAMP_Result_OK)
	-1: Error (Util64_TIMESTAMP_Result_Error)
	-2: DateValue Overflow (Util64_TIMESTAMP_Result_Overflow)
******************************************************************************)
FUNCTION Util64_TIMESTAMP_TO_DATETIME : DINT
VAR_INPUT
	Timestamp : UTIL64_TIMESTAMP;
	DateTimeResult : POINTER TO UTIL64_DATETIME;
END_VAR
;
END_FUNCTION

(* POU Util64_TIMESTAMP_TO_ECTIME, ST *)
(******************************************************************************
Description: Converts from 64bit Timestamp to Ethercat DC-Time.    
Input:
  - Timestamp: 64bit Timestamp structure containing nanoseconds since year 1970
  - ECTimeResult: 
    pointer to Ethercat 64bit Timestamp structure result containing nanoseconds
    since year 2000
Output:
    none
Return: DINT
	 0: Success (Util64_TIMESTAMP_Result_OK)
	-1: Error (Util64_TIMESTAMP_Result_Error)
	-3: Underflow as Timestamp < year 2000 (Util64_TIMESTAMP_Result_Underflow)
******************************************************************************)
FUNCTION Util64_TIMESTAMP_TO_ECTIME : DINT
VAR_INPUT
	Timestamp : UTIL64_TIMESTAMP;
	ECTimeResult : POINTER TO UTIL64_TIMESTAMP;
END_VAR
;
END_FUNCTION

(* POU Util64_TIMESTAMP_TO_LREAL, ST *)
(******************************************************************************
Description: Converts from unsigned 64bit Timestamp to LREAL.    
Input:
  - TimestampNs: 64bit Timestamp structure as nanoseconds
Output:
    none
Return:
	double float containing nanoseconds, the last digits can change due to 
    floating point arithmetic approximation.
    -1.0 on Error (NULL pointer)
******************************************************************************)
FUNCTION Util64_TIMESTAMP_TO_LREAL : LREAL
VAR_INPUT
	TimestampNs : UTIL64_TIMESTAMP;
END_VAR
;
END_FUNCTION

(* POU Util64_TIMESTAMP_TO_TIMESPEC, ST *)
(******************************************************************************
Description: Converts from 64bit Timestamp to TIMESPEC structure.    
Input:
  - TimestampNs: 64bit Timestamp structure as nanoseconds
  - TimespecResult: pointer to result TIMESPEC structure
Output:
    none
Return: DINT
	 0: Success (Util64_TIMESTAMP_Result_OK)
	-1: Error (Util64_TIMESTAMP_Result_Error)
	-2: Timespec.DATEANDTIME Overflow (Util64_TIMESTAMP_Result_Overflow)
******************************************************************************)
FUNCTION Util64_TIMESTAMP_TO_TIMESPEC : DINT
VAR_INPUT
	TimestampNs : UTIL64_TIMESTAMP;
	TimespecResult : POINTER TO TIMESPEC;
END_VAR
;
END_FUNCTION

(* POU Util_AddInt, IL *)
(******************************************************************************
Description: Appends an integer value to String
Input:
  - Str: Source String
  - Val: Value which is added to the end of the string
Output:
	none
Return:
  - String with the added value 
******************************************************************************)
FUNCTION Util_AddInt : STRING(255)
VAR_INPUT
	Str: STRING(255);
	Val: DWORD;
END_VAR
LD 0
END_FUNCTION

(* POU Util_CallCFcn, ST *)
(******************************************************************************
Description: Call a native C function. 
    First you have to fetch a function handle. When this succeded you can 
    call this function.
 Note: Only Use this FB when you well know C-API of VxWorks and M-SYS. You 
    should also know the functionality of PLC (see also to refering 
	documentation).
Input:
 - Cmd...Command of FB, see Util_CMD_FunctionCall
 - Param1 - Param6...Parameters passed to native C function
 - FcnName...function name
Output:
 - State...State of FB, see Util_ERR_CallC....
 - FcnReturn...Return value of C function
******************************************************************************)
FUNCTION_BLOCK Util_CallCFcn
VAR_INPUT
	Cmd:			DWORD;
	Param1:			DINT;
	Param2:			DINT;
	Param3:			DINT;
	Param4:			DINT;
	Param5:			DINT;
	Param6:			DINT;
	FcnName:		STRING(79);
END_VAR
VAR_OUTPUT
	State:			DINT;
	FcnReturn:		DINT;
END_VAR
VAR
	FcnHandle:		DWORD;
END_VAR
(* Dummy Programm *)
IF Cmd = Util_CMD_GetFcnHandle THEN
	FcnHandle := 55;
	State := Util_ERR_CallC_HandleOk;
ELSIF Cmd = Util_CMD_CallCFcn THEN
	IF FcnHandle = 0 THEN
		State := Util_ERR_CallC_NoHandle;
	ELSE
		State := Util_ERR_CallC_HandleOk;
		FcnReturn := 1;
	END_IF
ELSE
	State := Util_ERR_CallC_InvalidCmd;
END_IF
END_FUNCTION_BLOCK

(* POU Util_CallCFcnEx, ST *)
(******************************************************************************
Description: Call a native C function. 
    
The extended version operates in two modes: 
    First mode: 
     - First you have to fetch a function handle. When this succeded you can 
       call this function (like Util_CallCFcn). 
    Second mode: 
     - overgive the function handle as an input-parameter and call the 
       c-function without fetching the function handle first. 

 Note: Only Use this FB when you well know C-API of VxWorks and M-SYS. You 
       should also know the functionality of PLC (see also to refering 
       documentation). 
Input:
 - Cmd...Command of FB, see Util_CMD_FunctionCall
 - Param1 - Param6...Parameters passed to native C function
 - FcnName...function name
 - FcnHandle...function handle of c-function
Output:
 - State...State of FB, see Util_ERR_CallC....
 - FcnReturn...Return value of C function
******************************************************************************)
FUNCTION_BLOCK Util_CallCFcnEx
VAR_INPUT
	Cmd:			DWORD;
	Param1:			DINT;
	Param2:			DINT;
	Param3:			DINT;
	Param4:			DINT;
	Param5:			DINT;
	Param6:			DINT;
	FcnName:		STRING(79);
	FcnHandle:		DWORD;
END_VAR
VAR_OUTPUT
	State:			DINT;
	FcnReturn:		DINT;
END_VAR
VAR
END_VAR
(* Dummy Programm *)
IF Cmd = Util_CMD_GetFcnHandle THEN
	FcnHandle := 55;
	State := Util_ERR_CallC_HandleOk;
ELSIF Cmd = Util_CMD_CallCFcn THEN
	IF FcnHandle = 0 THEN
		State := Util_ERR_CallC_NoHandle;
	ELSE
		State := Util_ERR_CallC_HandleOk;
		FcnReturn := 1;
	END_IF
ELSE
	State := Util_ERR_CallC_InvalidCmd;
END_IF
END_FUNCTION_BLOCK

(* POU Util_CallCFcnNB, ST *)
(******************************************************************************
Description: Call a native C function (non blocking) 
Note: Only Use this FB when you well know C-API of VxWorks and M-SYS. You 
      should also know the functionality of PLC (see also to refering 
	  documentation).
Input:
 - Execute   Start execution of the function
 - FcnName   function name to call
 - FcnHandle if you haeve the handle (address) of the function provide
             this paramater instead of FcnName
 - Param1 - Param9  Parameters passed to native C function
 - Mode      Call native C funtion or PLC function (see Util_CallC_Mode_XXX)

Output:
 - FcnReturn Returned value of the ative C function called
 - Done      The execution of the FB is successfully finished
 - Busy      The execution of the FB is still in progress
 - Error     An error occured on execution of the FB
 - ErrorID   Errorcode (Util_ERR_CallC_XXX)

******************************************************************************)

FUNCTION_BLOCK Util_CallCFcnNB
VAR_INPUT
	Execute:	 BOOL;
	FcnName:	 STRING(79);
	FcnHandle:	 DWORD;
	Param1:      DINT;
	Param2:      DINT;
	Param3:      DINT;
	Param4:      DINT;
	Param5:      DINT;
	Param6:      DINT;
	Param7:      DINT;
	Param8:      DINT;
	Param9:      DINT;
	Mode:		 DINT;
END_VAR
VAR_OUTPUT
	FcnReturn:	 DINT;
	Done:	     BOOL;
	Busy:	     BOOL;
	Error: 		 BOOL;
	ErrorID: 	 DINT;
END_VAR
VAR
	pLTD:        DWORD;
	ExecuteM:	 BOOL;
END_VAR
;
END_FUNCTION_BLOCK

(* POU Util_Chr, IL *)
(******************************************************************************
Description: Converts the ASCII-Code to a string
Input:
  - Chr: Value, which represent the ASCII-Code
Output:
	none
Return: 
  - Character(String) of the ASCII-Code
******************************************************************************)
FUNCTION Util_Chr : STRING(1)
VAR_INPUT
	Chr: BYTE;
END_VAR
LD 0
END_FUNCTION

(* POU Util_DT_TO_TM, IL *)
(******************************************************************************
Description: Converts DT time to UTIL_TM (broken down time), without timezone 
             consideration. This routine performs the reverse translation that 
             UTIL_TM_TO_DT() does.
Input:
  - DateAndTime: Date and Time in DT format
Output:
    none
Return: 
    Date and Time in UTIL_TM format
******************************************************************************)
FUNCTION Util_DT_TO_TM: UTIL_TM
VAR_INPUT
    DateAndTime: DATE_AND_TIME;
END_VAR
	LD		0
END_FUNCTION

(* POU Util_DT_TO_TM_NB, ST *)
(******************************************************************************
Description: This is the non-blocking version of the function Util_DT_TO_TM().
             For further documentation see Util_DT_TO_TM().
Input:
  - DateAndTime: Date and Time in DT format
Output:
    none
Return: 
    Date and Time in UTIL_TM format
******************************************************************************)
FUNCTION_BLOCK Util_DT_TO_TM_NB
VAR_INPUT
    REQ : BOOL;
	DATEANDTIME: DATE_AND_TIME;
END_VAR
VAR_OUTPUT
	DONE : BOOL;
	ERROR : BOOL;
	STATUS : DINT;
	DateAndTimeTm: UTIL_TM;
END_VAR
VAR
    PLTD : DWORD;
END_VAR
;
END_FUNCTION_BLOCK

(* POU Util_ErrorString, IL *)
(******************************************************************************
Description: Get a short descriptive string to an ErrorCode
    (useful for ErrorCodes of SMI_PLC-Library)
Input:
  - Code: Errorcode
Output:
	none
Return: 
  - Errorstring
******************************************************************************)
FUNCTION Util_ErrorString : STRING(255)
VAR_INPUT
	Code: DINT;
END_VAR
LD 0
END_FUNCTION

(* POU Util_GetClock, ST *)
(******************************************************************************
Description: Gets the system clock value, using the system function 
             clock_gettime()
Input:
  - Source:  see VAR_CONSTANT Util_CLOCK_XXX
Output:
    none
Return:
  - TIMESPEC structure
******************************************************************************)
FUNCTION Util_GetClock : TIMESPEC
VAR_INPUT
	Source: DINT;
END_VAR
VAR
END_VAR
;
END_FUNCTION

(* POU Util_GetClockMonotonic, ST *)
(******************************************************************************
Description: Get a monotonous time from a specified time older than the start 
             of the system. This time is guaranteed to be monotonous even if 
             the "wall clock" time goes back.
Input:
  - Dummy: Parameter is not used
Output:
    none
Return:
  - TIMESPEC structure
******************************************************************************)
FUNCTION Util_GetClockMonotonic : TIMESPEC
VAR_INPUT
	Dummy: DINT;
END_VAR
VAR
END_VAR
;
END_FUNCTION

(* POU Util_GetCoreIndex, ST *)
(******************************************************************************
Description: Get the core index of the calling task. 
             Needs MSYS >= 4.30 R
Input:
  - pCoreIndex: The logical index is a number between 0 and N-1, where N is 
                the num-ber of CPUs configured in the MMP system. Calling this 
                function in the uniprocessor version of VxWorks returns 0, 
                always. 
Return: 
  - 0: OK
  - Tcs_ERC_NoSelf: is not a PLC project 
  - Tcs_ERC_Internal: not supported by MSYS
******************************************************************************)
FUNCTION Util_GetCoreIndex : DINT
VAR_INPUT
	pCoreIndex: POINTER TO UDINT;
END_VAR
VAR
END_VAR
;
END_FUNCTION

(* POU Util_GetCycStat, ST *)
(******************************************************************************
Description: Gets cycle-time- and run-time statistics/settings of the calling 
             task. The MSYS run-time measurement must be activated. 
             Needs MSYS >= 3.80 R
             
Input:
  - Dummy: meaningless
Output:
    none
Return:
  - UTIL_CYCSTAT structure
  - UTIL_CYCSTAT.ErrorCode: 
    - 0: OK
    - Tcs_ERC_Internal: not supported by MSYS or MSYS run-time measurement is 
                        not activated. 
******************************************************************************)
FUNCTION Util_GetCycStat : UTIL_CYCSTAT
VAR_INPUT
	Dummy: DINT;
END_VAR
VAR
END_VAR
;
END_FUNCTION

(* POU Util_GetProcTime, IL *)
(******************************************************************************
Description: Gets the current system timer
Input:
  - Dummy: Parameter is not used
Output:
    none
Return: 
    Elaspsed microseconds since boot (overrun every 1.2 hours)
******************************************************************************)
FUNCTION Util_GetProcTime : UDINT
VAR_INPUT
    Dummy: DINT;
END_VAR
LD FALSE
END_FUNCTION

(* POU Util_GetSymValByName, ST *)
(************************************************************************************
Description: get the value of a symbol in the vxworks symbol-table
Note: see the definition of a symbol in the MSYS header/include-files
      for a correct behaviour of this FB

Input:
 - Name ... a symbols name (the prefix "_" is added automatically)
 - Length ... length in Bytes of the symbols-value

Output:
 - Value ... the symbols-value
 - State ... possible errors (see global Util_ERR_SymVal_ constants), zero otherwise
************************************************************************************)
FUNCTION_BLOCK Util_GetSymValByName
VAR_INPUT
	Name: STRING(79);
	Length: USINT;
END_VAR
VAR_OUTPUT
	Value: UDINT;
	State: INT;
END_VAR
VAR
	SymHandle:	DWORD;
END_VAR
;
END_FUNCTION_BLOCK

(* POU Util_GetTimeZone, ST *)
(******************************************************************************
Description: Get the system timezone.

Input:
  - TimeZone: System timezone
Output:
  - TimeZone: 
Return:
  - Timezone offset in seconds to UTC
******************************************************************************)
FUNCTION Util_GetTimeZone : DINT
VAR_INPUT
	TimeZone: STRING;
END_VAR
VAR
END_VAR
;
END_FUNCTION

(* POU Util_GetUTCOffset, ST *)
(******************************************************************************
Description: Gets the actual timzone offset in seconds to UTC
Input:
  - Dummy Parameter is not used
Output:
    none
Return: 
	Actual time zone offset [s]
******************************************************************************)
FUNCTION Util_GetUTCOffset : DINT
VAR_INPUT
	Dummy: BOOL;
END_VAR
VAR
END_VAR
;
END_FUNCTION

(* POU Util_GetVersion, ST *)
(******************************************************************************
Description: Returns the version string of the library. In simulation always
	'' is returned.

Input:
	- dummy

Return: 
	Version String
******************************************************************************)
FUNCTION Util_GetVersion : STRING(15)
VAR_INPUT
	dummy:		BOOL;
END_VAR
VAR
END_VAR
Util_GetVersion := '';
END_FUNCTION

(* POU Util_LIST_Create, ST *)
(******************************************************************************
Description: Create a list. 

Input:
 - ElemSize...Size of one element in the list
 - ListLen...length of the list

Output:
 - Handle...Handle of list. Use it at other functions.
 - State...0 - List was created
           <0 - Error occured, see Util_ERR_Lst....
******************************************************************************)
FUNCTION_BLOCK Util_LIST_Create
VAR_INPUT
	ElemSize:		DINT;
	ListLen:		DINT;
END_VAR
VAR_OUTPUT
	Handle:			DWORD;
	State:			DINT;
END_VAR
VAR
END_VAR
;
END_FUNCTION_BLOCK

(* POU Util_LIST_Get, ST *)
(******************************************************************************
Description: Get a element of a list. Element is copied into buffer.

Input:
 - Handle...Handle of list
 - DataAdr...Address of buffer. Into this buffer element content is copied,
       use ADR()
 - DataLen...Length of buffer
 - Mode...Mode of getting a list element, see Util_LIST_Getxxx
 - FindId...Element ID to find at mode Util_LIST_GetById

Output:
 - ElemId...Element Id of element
 - CopySize...Size of copied data
 - State...0 - Element was found
           <0 - Error occured, see Util_ERR_Lst....
******************************************************************************)
FUNCTION_BLOCK Util_LIST_Get
VAR_INPUT
	Handle:			DWORD;
	DataAddr:		DWORD;
	DataLen:		DINT;
	Mode:			DINT;
	FindId:			DWORD;
END_VAR
VAR_OUTPUT
	ElemId:			DWORD;
	CopySize:		DINT;
	State:			DINT;
END_VAR
VAR
END_VAR
;
END_FUNCTION_BLOCK

(* POU Util_LIST_Insert, ST *)
(******************************************************************************
Description: Insert a element into the list. The element content is
	 copied into the list.
  Note: At most ElemSize (parameter of Util_LISTCreate) is copied into the list.
    If DataLen is bigger, the enty is shortend in the list.

Input:
 - Handle...Handle of list
 - DataAddr...Address of data buffer, use ADR()
 - DataLen...Length of data buffer
 - Mode...Mode of insert a list element, see Util_LIST_Insertxxx

Output:
 - ElemId...Id of list element 
 - CopySize...Copied size 
 - State...0 - Element was inserted to list
           <0 - Error occured, see Util_ERR_Lst....
******************************************************************************)
FUNCTION_BLOCK Util_LIST_Insert
VAR_INPUT
	Handle:			DWORD;
	DataAddr:		DWORD;
	DataLen:		DINT;
	Mode:			DINT;
END_VAR
VAR_OUTPUT
	ElemId:			UDINT;
	CopySize:		DINT;
	State:			DINT;
END_VAR
VAR
END_VAR
;
END_FUNCTION_BLOCK

(* POU Util_LIST_Remove, ST *)
(******************************************************************************
Description: Remove a element or all elements of a list. 

Input:
 - Handle...handle of list
 - Mode...Where element is added, see Util_LIST_Removexxx

Output:
 - ElemId...Id of removed list element 
 - State...0 - Element was removed
           <0 - Error occured, see Util_ERR_Lst....
******************************************************************************)
FUNCTION_BLOCK Util_LIST_Remove
VAR_INPUT
	Handle:			DWORD;
	Mode:			DINT;
END_VAR
VAR_OUTPUT
	ElemId:			UDINT;
	State:			DINT;
END_VAR
VAR
END_VAR
;
END_FUNCTION_BLOCK

(* POU Util_LogErr, IL *)
(******************************************************************************
Description: Write message as Error ("E:...") to logbook and console
Input:
  - Str: Message-String
Output:
	none
Return: Meaningless
******************************************************************************)
FUNCTION Util_LogErr : DINT
VAR_INPUT
	Str: STRING(255);
END_VAR
	LD		0
END_FUNCTION

(* POU Util_LogInfo, IL *)
(******************************************************************************
Description: Write message as Info ("I:...") to logbook and console
Input:
  - Str: Message-String
Output:
	none
Return: Meaningless
******************************************************************************)
FUNCTION Util_LogInfo : DINT
VAR_INPUT
	Str: STRING(255);
END_VAR
LD 0
END_FUNCTION

(* POU Util_LogSetDebugMode, ST *)
(******************************************************************************
Description: This functions sets the Debug Mode of the logging functions.
			 If the DebugMode = TRUE Util_LogInfo and Util_LogWrn are printed
             only if the corresponding DebugLevel is set for the application.   
Input:
  - UseDebugMode: Flag if UseDebugMode shall be used
Output:
	none
Return: 0 on success, -1 on error
******************************************************************************)

FUNCTION Util_LogSetDebugMode : DINT
VAR_INPUT
	UseDebugMode: BOOL;
END_VAR
;
END_FUNCTION

(* POU Util_LogWrn, IL *)
(******************************************************************************
Description: Write message as Warning ("W:...") to logbook and console
Input:
  - Str: Message-String
Output:
	none
Return: Meaningless
******************************************************************************)
FUNCTION Util_LogWrn : DINT
VAR_INPUT
	Str: STRING(255);
END_VAR
LD 0
END_FUNCTION

(* POU Util_Ord, IL *)
(******************************************************************************
Description: Converts a character in the STRING to its BYTE-ASCII-Code
Input:
  - Str: Input Strint
  - Index: Index of the character; range from 1 to LEN 
Output:
	none
Return:
  - ASCII Code of the character
******************************************************************************)
FUNCTION Util_Ord : BYTE
VAR_INPUT
	Str: STRING(255);
	Index: DINT;
END_VAR
LD 0
END_FUNCTION

(* POU Util_RTC_GetDateAndTime, IL *)
(******************************************************************************
Description: Gets the current system date & time (UTC/LOCAL).
             This routine returns the current system time in either UTC or 
             LOCAL time representation, depending on given time mode.
Input:
  - Mode: Time Mode (see Util_DT_Mode_XXX)
Output:
    none
Return: 
    Current date and time of format DATE_AND_TIME 
******************************************************************************)
FUNCTION Util_RTC_GetDateAndTime: DATE_AND_TIME
VAR_INPUT
    Mode: DINT;
END_VAR
	LD		0
END_FUNCTION

(* POU Util_RTC_SetDateAndTime, IL *)
(******************************************************************************
Description: Sets the current system date & time.
             This routine sets the system clock to the time specified. Given
             time represents UTC or LOCAL time, depending on given time mode.
Input:
  - DatenAndTime: System date to set
  - Mode:         Time Mode (see Util_DT_Mode_XXX)
Output:
    none
Return: 
    Errorcode
******************************************************************************)
FUNCTION Util_RTC_SetDateAndTime: DINT
VAR_INPUT
	DateAndTime: DATE_AND_TIME;
    Mode: DINT;
END_VAR
	LD		0
END_FUNCTION

(* POU Util_SetCoreCategory, ST *)
(******************************************************************************
Description: Adjust the core category of the calling task. 
             Needs MSYS >= 4.30 R
Input:
  - CoreCategory: core category/affinity of task 
Return: 
  - 0: OK
  - Tcs_ERC_NoSelf: is not a PLC project 
  - Tcs_ERC_Internal: not supported by MSYS
  - Tcs_ERC_ParmInvalid: category is invalid 
******************************************************************************)
FUNCTION Util_SetCoreCategory : DINT
VAR_INPUT
	CoreCategory: STRING;
END_VAR
VAR
END_VAR
;
END_FUNCTION

(* POU Util_SetCycStat, ST *)
(******************************************************************************
Description: Adjusts cycle-time/task-related settings of the calling task. 
             Needs MSYS >= 3.80 R
Input:
  - CycTime: cycle-time [us]
  - MainRatio: execution-rate of the task-POU
  - Priority: VxWorks priority between 18 and 253
Output:
    none
Return: 
    - 0: OK
    - Tcs_ERC_Internal: not supported by MSYS
******************************************************************************)
FUNCTION Util_SetCycStat : DINT
VAR_INPUT
	CycTime: DWORD;
    MainRatio: DINT;
    Priority: DINT;
END_VAR
;
END_FUNCTION

(* POU Util_SetSymValByName, ST *)
(************************************************************************************
Description: set the value of a symbol in the vxworks symbol-table
Note: see the definition of a symbol in the MSYS header/include-files
      for a correct behaviour of this FB

Input:
 - Name ... a symbols name (the prefix "_" is added automatically)
 - Value ... symbols-value to set
 - Length ... length in Bytes of the symbols-value

Output:
 - State ... possible errors (see global Util_ERR_SymVal_ constants), zero otherwise
************************************************************************************)
FUNCTION_BLOCK Util_SetSymValByName
VAR_INPUT
	Name: STRING(79);
	Value: UDINT;
	Length: USINT;
END_VAR
VAR_OUTPUT
	State: INT;
END_VAR
VAR
	SymHandle:	DWORD;
END_VAR
;
END_FUNCTION_BLOCK

(* POU Util_SetTimeZone, ST *)
(******************************************************************************
Description: Sets the system timezone

Input:
  - TimeZone: New system timezone
  - Remanent: Set permanently (save to mconfig.ini)
Output:
  - TimeZone: 
Return:
    Errorcode

Since: MSYS V3.95
******************************************************************************)
FUNCTION Util_SetTimeZone : DINT
VAR_INPUT
	TimeZone: STRING;
    Remanent: BOOL;
END_VAR
VAR
END_VAR
;
END_FUNCTION

(* POU Util_TM_TO_DT, IL *)
(******************************************************************************
Description: Converts UTIL_TM (broken down time) to DT time, without timezone
             consideration. This routine performs the reverse translation that 
             UTIL_DT_TO_TM() does.
Input:
  - DateAndTime: Date and Time in UTIL_TM format
Output:
    none
Return: 
    Date and Time in DATE_AND_TIME format
******************************************************************************)
FUNCTION Util_TM_TO_DT: DATE_AND_TIME
VAR_INPUT
    DateAndTime: UTIL_TM;
END_VAR
	LD		0
END_FUNCTION

(* POU Util_TM_TO_DT_NB, ST *)
(******************************************************************************
Description: This is the non-blocking version of the function Util_TM_TO_DT().
             For further documentation see Util_TM_TO_DT().
Input:
  - DateAndTime: Date and Time in UTIL_TM format
Output:
    none
Return: 
    Date and Time in DATE_AND_TIME format
******************************************************************************)
FUNCTION_BLOCK Util_TM_TO_DT_NB
VAR_INPUT
    REQ : BOOL;
	DateAndTimeTm: UTIL_TM;
END_VAR
VAR_OUTPUT
	DONE : BOOL;
	ERROR : BOOL;
	STATUS : DINT;
	DateAndTime: DATE_AND_TIME;
END_VAR
VAR
	PLTD : DWORD;
END_VAR
;
END_FUNCTION_BLOCK
